  MoveL 5887 to (-63.75, 25.43, -226.45) mm, rotated rx -172.19 ry 6.28 rz 7.52 deg; joints [-6.092, -28.994, 83.557, 94.01, 104.935, 56.545, -36.259]
  MoveL 5888 to (-64.25, 25.28, -226.45) mm, rotated rx -172.19 ry 6.28 rz 7.52 deg; joints [-6.076, -29.01, 83.573, 94.023, 104.926, 56.543, -36.259]
  MoveL 5889 to (-65.23, 24.96, -226.41) mm, rotated rx -172.19 ry 6.28 rz 7.52 deg; joints [-6.045, -29.04, 83.608, 94.048, 104.908, 56.538, -36.259]
  MoveL 5890 to (-67.74, 24.21, -226.41) mm, rotated rx -172.19 ry 6.28 rz 7.52 deg; joints [-5.965, -29.118, 83.687, 94.111, 104.862, 56.533, -36.259]
  MoveL 5891 to (-68.71, 23.85, -226.39) mm, rotated rx -172.19 ry 6.28 rz 7.52 deg; joints [-5.934, -29.151, 83.725, 94.135, 104.844, 56.527, -36.259]
  MoveL 5892 to (-70.09, 23.42, -226.46) mm, rotated rx -172.19 ry 6.28 rz 7.52 deg; joints [-5.891, -29.197, 83.77, 94.17, 104.819, 56.527, -36.259]
  MoveL 5893 to (-71.24, 23.21, -226.71) mm, rotated rx -172.19 ry 6.28 rz 7.52 deg; joints [-5.856, -29.233, 83.787, 94.203, 104.798, 56.544, -36.259]
  MoveL 5894 to (-72.17, 23.22, -227.15) mm, rotated rx -172.19 ry 6.28 rz 7.52 deg; joints [-5.831, -29.259, 83.777, 94.232, 104.781, 56.579, -36.259]
  MoveL 5895 to (-72.55, 23.31, -227.44) mm, rotated rx -172.19 ry 6.28 rz 7.52 deg; joints [-5.822, -29.268, 83.763, 94.245, 104.774, 56.604, -36.259]
  MoveL 5896 to (-72.88, 23.45, -227.78) mm, rotated rx -172.19 ry 6.28 rz 7.52 deg; joints [-5.816, -29.274, 83.741, 94.258, 104.768, 56.632, -36.259]
  MoveL 5897 to (-73.35, 23.9, -228.59) mm, rotated rx -172.19 ry 6.28 rz 7.52 deg; joints [-5.809, -29.28, 83.677, 94.282, 104.759, 56.703, -36.259]
  MoveL 5898 to (-73.61, 24.57, -229.59) mm, rotated rx -172.19 ry 6.28 rz 7.52 deg; joints [-5.812, -29.275, 83.587, 94.302, 104.754, 56.792, -36.259]
  MoveL 5899 to (-73.44, 26.58, -232.15) mm, rotated rx -172.19 ry 6.28 rz 7.52 deg; joints [-5.844, -29.234, 83.324, 94.334, 104.756, 57.022, -36.259]
  MoveL 5900 to (-72.5, 28.79, -234.71) mm, rotated rx -172.19 ry 6.28 rz 7.52 deg; joints [-5.901, -29.171, 83.039, 94.347, 104.773, 57.254, -36.259]
  MoveL 5901 to (-70.94, 30.53, -236.54) mm, rotated rx -172.19 ry 6.28 rz 7.52 deg; joints [-5.97, -29.104, 82.818, 94.333, 104.802, 57.415, -36.259]
  MoveL 5902 to (-69.92, 31.22, -237.18) mm, rotated rx -172.19 ry 6.28 rz 7.52 deg; joints [-6.009, -29.069, 82.733, 94.316, 104.821, 57.469, -36.259]
  MoveL 5903 to (-68.75, 31.79, -237.64) mm, rotated rx -172.19 ry 6.28 rz 7.52 deg; joints [-6.051, -29.034, 82.664, 94.291, 104.843, 57.506, -36.259]
  MoveL 5904 to (-65.94, 32.57, -238.01) mm, rotated rx -172.19 ry 6.28 rz 7.52 deg; joints [-6.144, -28.962, 82.575, 94.221, 104.897, 57.527, -36.259]
  MoveL 5905 to (-62.84, 33.11, -238.01) mm, rotated rx -172.19 ry 6.28 rz 7.52 deg; joints [-6.243, -28.889, 82.52, 94.139, 104.957, 57.514, -36.259]
  MoveL 5906 to (-61.85, 33.31, -238.02) mm, rotated rx -172.19 ry 6.28 rz 7.52 deg; joints [-6.274, -28.865, 82.499, 94.113, 104.976, 57.511, -36.259]
  MoveL 5907 to (-60.81, 33.49, -238.02) mm, rotated rx -172.19 ry 6.28 rz 7.52 deg; joints [-6.307, -28.84, 82.48, 94.085, 104.996, 57.507, -36.259]
  MoveL 5908 to (-60.32, 33.58, -238.02) mm, rotated rx -172.19 ry 6.28 rz 7.52 deg; joints [-6.323, -28.829, 82.471, 94.072, 105.005, 57.505, -36.259]
  MoveL 5909 to (-59.67, 33.7, -238.05) mm, rotated rx -172.19 ry 6.28 rz 7.52 deg; joints [-6.344, -28.814, 82.457, 94.055, 105.018, 57.505, -36.259]
  MoveL 5910 to (-59.09, 33.84, -238.11) mm, rotated rx -172.19 ry 6.28 rz 7.52 deg; joints [-6.363, -28.8, 82.443, 94.04, 105.029, 57.507, -36.259]
  MoveL 5911 to (-58.6, 33.97, -238.18) mm, rotated rx -172.19 ry 6.28 rz 7.52 deg; joints [-6.379, -28.788, 82.427, 94.028, 105.038, 57.511, -36.259]
  MoveL 5912 to (-58.15, 34.08, -238.24) mm, rotated rx -172.19 ry 6.28 rz 7.52 deg; joints [-6.394, -28.777, 82.414, 94.017, 105.047, 57.513, -36.259]
  MoveL 5913 to (-57.7, 34.18, -238.27) mm, rotated rx -172.19 ry 6.28 rz 7.52 deg; joints [-6.409, -28.766, 82.403, 94.005, 105.055, 57.514, -36.259]
  MoveL 5914 to (-56.15, 34.45, -238.27) mm, rotated rx -172.19 ry 6.28 rz 7.52 deg; joints [-6.458, -28.729, 82.375, 93.964, 105.085, 57.508, -36.259]
  MoveL 5915 to (-55.66, 34.56, -238.28) mm, rotated rx -172.19 ry 6.28 rz 7.52 deg; joints [-6.473, -28.716, 82.363, 93.951, 105.094, 57.507, -36.259]
  MoveL 5916 to (-55.23, 34.67, -238.31) mm, rotated rx -172.19 ry 6.28 rz 7.52 deg; joints [-6.487, -28.705, 82.35, 93.941, 105.102, 57.509, -36.259]
  MoveL 5917 to (-54.87, 34.8, -238.36) mm, rotated rx -172.19 ry 6.28 rz 7.52 deg; joints [-6.499, -28.693, 82.335, 93.932, 105.109, 57.514, -36.259]
  MoveL 5918 to (-54.61, 34.96, -238.42) mm, rotated rx -172.19 ry 6.28 rz 7.52 deg; joints [-6.508, -28.682, 82.316, 93.927, 105.114, 57.522, -36.259]
  MoveL 5919 to (-54.41, 35.14, -238.49) mm, rotated rx -172.19 ry 6.28 rz 7.52 deg; joints [-6.515, -28.671, 82.295, 93.924, 105.118, 57.532, -36.259]
  MoveL 5920 to (-55.91, 34.64, -239.3) mm, rotated rx -172.19 ry 6.28 rz 7.52 deg; joints [-6.476, -28.747, 82.338, 93.964, 105.092, 57.565, -36.259]
  MoveL 5921 to (-54.61, 35.83, -239.7) mm, rotated rx -172.19 ry 6.28 rz 7.52 deg; joints [-6.521, -28.669, 82.197, 93.945, 105.115, 57.632, -36.259]
  MoveL 5922 to (-53.25, 37.12, -239.96) mm, rotated rx -172.19 ry 6.28 rz 7.52 deg; joints [-6.566, -28.581, 82.047, 93.926, 105.137, 57.697, -36.259]
  MoveL 5923 to (-51.81, 38.51, -240.15) mm, rotated rx -172.19 ry 6.28 rz 7.52 deg; joints [-6.612, -28.481, 81.886, 93.906, 105.16, 57.763, -36.259]
  MoveL 5924 to (-50.29, 40.01, -240.34) mm, rotated rx -172.19 ry 6.28 rz 7.52 deg; joints [-6.661, -28.375, 81.712, 93.886, 105.185, 57.835, -36.259]
  MoveL 5925 to (-48.76, 41.5, -240.44) mm, rotated rx -172.19 ry 6.28 rz 7.52 deg; joints [-6.709, -28.265, 81.541, 93.865, 105.209, 57.901, -36.259]
  MoveL 5926 to (-47.23, 42.98, -240.53) mm, rotated rx -172.19 ry 6.28 rz 7.52 deg; joints [-6.757, -28.156, 81.369, 93.844, 105.234, 57.967, -36.259]
  MoveL 5927 to (-45.7, 44.48, -240.73) mm, rotated rx -172.19 ry 6.28 rz 7.52 deg; joints [-6.806, -28.049, 81.194, 93.824, 105.258, 58.04, -36.259]
  MoveL 5928 to (-44.17, 45.96, -240.83) mm, rotated rx -172.19 ry 6.28 rz 7.52 deg; joints [-6.854, -27.939, 81.022, 93.803, 105.283, 58.107, -36.259]
  MoveL 5929 to (-42.63, 47.44, -240.93) mm, rotated rx -172.19 ry 6.28 rz 7.52 deg; joints [-6.902, -27.83, 80.849, 93.782, 105.307, 58.174, -36.259]
  MoveL 5930 to (-41.09, 48.92, -241.13) mm, rotated rx -172.19 ry 6.28 rz 7.52 deg; joints [-6.951, -27.723, 80.674, 93.763, 105.332, 58.247, -36.259]
  MoveL 5931 to (-38.01, 51.88, -241.33) mm, rotated rx -172.19 ry 6.28 rz 7.52 deg; joints [-7.046, -27.503, 80.326, 93.722, 105.382, 58.383, -36.259]
  MoveL 5932 to (-36.72, 53.11, -241.54) mm, rotated rx -172.19 ry 6.28 rz 7.52 deg; joints [-7.088, -27.414, 80.178, 93.706, 105.403, 58.446, -36.259]
  MoveL 5933 to (-35.33, 54.5, -241.61) mm, rotated rx -172.19 ry 6.28 rz 7.52 deg; joints [-7.131, -27.31, 80.014, 93.689, 105.425, 58.51, -36.259]
  MoveL 5934 to (-33.91, 55.99, -241.62) mm, rotated rx -172.19 ry 6.28 rz 7.52 deg; joints [-7.173, -27.197, 79.838, 93.673, 105.447, 58.577, -36.259]
  MoveL 5935 to (-31.97, 57.83, -241.73) mm, rotated rx -172.19 ry 6.28 rz 7.52 deg; joints [-7.233, -27.058, 79.619, 93.648, 105.478, 58.662, -36.259]
  MoveL 5936 to (-30.02, 59.52, -241.83) mm, rotated rx -172.19 ry 6.28 rz 7.52 deg; joints [-7.293, -26.928, 79.417, 93.621, 105.509, 58.739, -36.259]
  MoveL 5937 to (-28.4, 61.01, -241.92) mm, rotated rx -172.19 ry 6.28 rz 7.52 deg; joints [-7.343, -26.814, 79.237, 93.6, 105.536, 58.809, -36.259]
  MoveL 5938 to (-26.9, 62.41, -242.1) mm, rotated rx -172.19 ry 6.28 rz 7.52 deg; joints [-7.39, -26.71, 79.067, 93.582, 105.56, 58.879, -36.259]
  MoveL 5939 to (-25.5, 63.7, -242.38) mm, rotated rx -172.19 ry 6.28 rz 7.52 deg; joints [-7.435, -26.617, 78.908, 93.565, 105.583, 58.95, -36.259]
  MoveL 5940 to (-24.11, 64.98, -242.66) mm, rotated rx -172.19 ry 6.28 rz 7.52 deg; joints [-7.479, -26.525, 78.749, 93.549, 105.607, 59.021, -36.259]
  MoveL 5941 to (-22.7, 66.23, -242.96) mm, rotated rx -172.19 ry 6.28 rz 7.52 deg; joints [-7.525, -26.436, 78.594, 93.532, 105.63, 59.09, -36.259]
  MoveL 5942 to (-21.23, 67.57, -243.11) mm, rotated rx -172.19 ry 6.28 rz 7.52 deg; joints [-7.57, -26.334, 78.429, 93.514, 105.654, 59.158, -36.259]
  MoveL 5943 to (-20.58, 67.57, -243.73) mm, rotated rx -172.19 ry 6.28 rz 7.52 deg; joints [-7.597, -26.345, 78.42, 93.499, 105.67, 59.18, -36.259]
  MoveL 5944 to (-20.69, 67.27, -244.04) mm, rotated rx -172.19 ry 6.28 rz 7.52 deg; joints [-7.598, -26.375, 78.451, 93.498, 105.67, 59.179, -36.259]
  MoveL 5945 to (-20.66, 67.23, -244.24) mm, rotated rx -172.19 ry 6.28 rz 7.52 deg; joints [-7.601, -26.383, 78.453, 93.498, 105.671, 59.186, -36.259]
  MoveL 5946 to (-20.52, 67.44, -244.33) mm, rotated rx -172.19 ry 6.28 rz 7.52 deg; joints [-7.606, -26.371, 78.426, 93.498, 105.674, 59.201, -36.259]
  MoveL 5947 to (-20.34, 67.85, -244.35) mm, rotated rx -172.19 ry 6.28 rz 7.52 deg; joints [-7.611, -26.343, 78.376, 93.5, 105.675, 59.223, -36.259]
  MoveL 5948 to (-20.18, 68.31, -244.36) mm, rotated rx -172.19 ry 6.28 rz 7.52 deg; joints [-7.615, -26.311, 78.321, 93.503, 105.676, 59.248, -36.259]
  MoveL 5949 to (-19.97, 69.26, -244.39) mm, rotated rx -172.19 ry 6.28 rz 7.52 deg; joints [-7.621, -26.248, 78.205, 93.514, 105.677, 59.303, -36.259]
  MoveL 5950 to (-19.63, 70.8, -244.39) mm, rotated rx -172.19 ry 6.28 rz 7.52 deg; joints [-7.629, -26.144, 78.019, 93.53, 105.677, 59.388, -36.259]
  MoveL 5951 to (-19.38, 71.74, -244.4) mm, rotated rx -172.19 ry 6.28 rz 7.52 deg; joints [-7.635, -26.081, 77.904, 93.54, 105.677, 59.441, -36.259]
  MoveL 5952 to (-19.16, 72.77, -244.4) mm, rotated rx -172.19 ry 6.28 rz 7.52 deg; joints [-7.64, -26.011, 77.78, 93.551, 105.677, 59.499, -36.259]
  MoveL 5953 to (-19.04, 73.27, -244.42) mm, rotated rx -172.19 ry 6.28 rz 7.52 deg; joints [-7.643, -25.978, 77.719, 93.557, 105.677, 59.528, -36.259]
  MoveL 5954 to (-18.93, 73.73, -244.45) mm, rotated rx -172.19 ry 6.28 rz 7.52 deg; joints [-7.646, -25.948, 77.663, 93.561, 105.678, 59.554, -36.259]
  MoveL 5955 to (-18.81, 74.15, -244.49) mm, rotated rx -172.19 ry 6.28 rz 7.52 deg; joints [-7.65, -25.92, 77.611, 93.566, 105.678, 59.58, -36.259]
  MoveL 5956 to (-18.7, 74.54, -244.56) mm, rotated rx -172.19 ry 6.28 rz 7.52 deg; joints [-7.653, -25.895, 77.562, 93.569, 105.679, 59.605, -36.259]
  MoveL 5957 to (-18.58, 74.94, -244.61) mm, rotated rx -172.19 ry 6.28 rz 7.52 deg; joints [-7.657, -25.869, 77.512, 93.573, 105.68, 59.63, -36.259]
  MoveL 5958 to (-18.46, 75.39, -244.64) mm, rotated rx -172.19 ry 6.28 rz 7.52 deg; joints [-7.66, -25.84, 77.457, 93.578, 105.68, 59.656, -36.259]
  MoveL 5959 to (-18.35, 75.85, -244.67) mm, rotated rx -172.19 ry 6.28 rz 7.52 deg; joints [-7.663, -25.809, 77.4, 93.583, 105.68, 59.683, -36.259]
  MoveL 5960 to (-18.22, 76.27, -244.71) mm, rotated rx -172.19 ry 6.28 rz 7.52 deg; joints [-7.667, -25.781, 77.349, 93.587, 105.681, 59.709, -36.259]
  MoveL 5961 to (-18.1, 76.65, -244.77) mm, rotated rx -172.19 ry 6.28 rz 7.52 deg; joints [-7.671, -25.757, 77.301, 93.59, 105.682, 59.733, -36.259]
  MoveL 5962 to (-17.98, 77.04, -244.82) mm, rotated rx -172.19 ry 6.28 rz 7.52 deg; joints [-7.674, -25.731, 77.252, 93.594, 105.683, 59.757, -36.259]
  MoveL 5963 to (-17.86, 77.47, -244.85) mm, rotated rx -172.19 ry 6.28 rz 7.52 deg; joints [-7.678, -25.703, 77.2, 93.598, 105.683, 59.782, -36.259]
  MoveL 5964 to (-17.75, 77.98, -244.85) mm, rotated rx -172.19 ry 6.28 rz 7.52 deg; joints [-7.68, -25.668, 77.137, 93.604, 105.683, 59.811, -36.259]
  MoveL 5965 to (-16.88, 80.76, -245.21) mm, rotated rx -172.19 ry 6.28 rz 7.52 deg; joints [-7.707, -25.485, 76.79, 93.63, 105.689, 59.983, -36.259]
  MoveL 5966 to (-16.3, 81.92, -245.65) mm, rotated rx -172.19 ry 6.28 rz 7.52 deg; joints [-7.727, -25.416, 76.64, 93.637, 105.697, 60.067, -36.259]
  MoveL 5967 to (-15.62, 82.91, -246.28) mm, rotated rx -172.19 ry 6.28 rz 7.52 deg; joints [-7.753, -25.36, 76.507, 93.639, 105.708, 60.148, -36.259]
  MoveL 5968 to (-13.99, 84.42, -248.06) mm, rotated rx -172.19 ry 6.28 rz 7.52 deg; joints [-7.82, -25.293, 76.29, 93.629, 105.741, 60.306, -36.259]
  MoveL 5969 to (-11.99, 85.29, -250.55) mm, rotated rx -172.19 ry 6.28 rz 7.52 deg; joints [-7.907, -25.283, 76.139, 93.603, 105.786, 60.456, -36.259]
  MoveL 5970 to (-10.19, 85.39, -253.05) mm, rotated rx -172.19 ry 6.28 rz 7.52 deg; joints [-7.988, -25.326, 76.082, 93.569, 105.832, 60.563, -36.259]
  MoveL 5971 to (-9.6, 85.11, -254.02) mm, rotated rx -172.19 ry 6.28 rz 7.52 deg; joints [-8.017, -25.365, 76.099, 93.553, 105.849, 60.587, -36.259]
  MoveL 5972 to (-9.2, 84.61, -254.83) mm, rotated rx -172.19 ry 6.28 rz 7.52 deg; joints [-8.039, -25.417, 76.147, 93.538, 105.862, 60.592, -36.259]
  MoveL 5973 to (-9.08, 84.28, -255.16) mm, rotated rx -172.19 ry 6.28 rz 7.52 deg; joints [-8.047, -25.447, 76.183, 93.53, 105.867, 60.587, -36.259]
  MoveL 5974 to (-9.01, 83.89, -255.45) mm, rotated rx -172.19 ry 6.28 rz 7.52 deg; joints [-8.052, -25.48, 76.226, 93.523, 105.872, 60.577, -36.259]
  MoveL 5975 to (-9.02, 82.94, -255.89) mm, rotated rx -172.19 ry 6.28 rz 7.52 deg; joints [-8.059, -25.556, 76.335, 93.509, 105.877, 60.542, -36.259]
  MoveL 5976 to (-9.23, 81.77, -256.16) mm, rotated rx -172.19 ry 6.28 rz 7.52 deg; joints [-8.057, -25.644, 76.475, 93.495, 105.88, 60.488, -36.259]
  MoveL 5977 to (-9.65, 80.38, -256.25) mm, rotated rx -172.19 ry 6.28 rz 7.52 deg; joints [-8.048, -25.744, 76.645, 93.482, 105.878, 60.414, -36.259]
  MoveL 5978 to (-10.5, 77.9, -256.25) mm, rotated rx -172.19 ry 6.28 rz 7.52 deg; joints [-8.026, -25.918, 76.951, 93.462, 105.872, 60.277, -36.259]
  MoveL 5979 to (-10.65, 77.49, -256.22) mm, rotated rx -172.19 ry 6.28 rz 7.52 deg; joints [-8.021, -25.946, 77.002, 93.458, 105.871, 60.253, -36.259]
  MoveL 5980 to (-10.81, 77.12, -256.17) mm, rotated rx -172.19 ry 6.28 rz 7.52 deg; joints [-8.017, -25.971, 77.048, 93.456, 105.869, 60.231, -36.259]
  MoveL 5981 to (-10.97, 76.77, -256.1) mm, rotated rx -172.19 ry 6.28 rz 7.52 deg; joints [-8.012, -25.994, 77.093, 93.454, 105.867, 60.208, -36.259]
  MoveL 5982 to (-11.13, 76.37, -256.05) mm, rotated rx -172.19 ry 6.28 rz 7.52 deg; joints [-8.007, -26.021, 77.142, 93.451, 105.866, 60.184, -36.259]
  MoveL 5983 to (-11.31, 75.9, -256.01) mm, rotated rx -172.19 ry 6.28 rz 7.52 deg; joints [-8.002, -26.053, 77.2, 93.447, 105.864, 60.157, -36.259]
  MoveL 5984 to (-11.51, 75.42, -255.96) mm, rotated rx -172.19 ry 6.28 rz 7.52 deg; joints [-7.996, -26.085, 77.261, 93.444, 105.862, 60.128, -36.259]
  MoveL 5985 to (-11.69, 74.91, -255.94) mm, rotated rx -172.19 ry 6.28 rz 7.52 deg; joints [-7.991, -26.121, 77.324, 93.44, 105.861, 60.099, -36.259]
  MoveL 5986 to (-11.9, 74.3, -255.96) mm, rotated rx -172.19 ry 6.28 rz 7.52 deg; joints [-7.986, -26.163, 77.398, 93.435, 105.859, 60.067, -36.259]
  MoveL 5987 to (-12.15, 73.47, -256.02) mm, rotated rx -172.19 ry 6.28 rz 7.52 deg; joints [-7.98, -26.223, 77.498, 93.428, 105.858, 60.024, -36.259]
  MoveL 5988 to (-12.32, 72.97, -256.02) mm, rotated rx -172.19 ry 6.28 rz 7.52 deg; joints [-7.976, -26.258, 77.558, 93.424, 105.857, 59.997, -36.259]
  MoveL 5989 to (-12.49, 72.5, -256.01) mm, rotated rx -172.19 ry 6.28 rz 7.52 deg; joints [-7.971, -26.29, 77.616, 93.42, 105.856, 59.971, -36.259]
  MoveL 5990 to (-12.65, 72.06, -255.99) mm, rotated rx -172.19 ry 6.28 rz 7.52 deg; joints [-7.967, -26.32, 77.67, 93.417, 105.854, 59.947, -36.259]
  MoveL 5991 to (-12.81, 71.68, -255.94) mm, rotated rx -172.19 ry 6.28 rz 7.52 deg; joints [-7.962, -26.346, 77.717, 93.415, 105.853, 59.924, -36.259]
  MoveL 5992 to (-12.98, 71.32, -255.88) mm, rotated rx -172.19 ry 6.28 rz 7.52 deg; joints [-7.957, -26.37, 77.762, 93.413, 105.851, 59.902, -36.259]
  MoveL 5993 to (-13.2, 70.96, -255.83) mm, rotated rx -172.19 ry 6.28 rz 7.52 deg; joints [-7.95, -26.395, 77.807, 93.412, 105.848, 59.881, -36.259]
  MoveL 5994 to (-13.45, 70.63, -255.78) mm, rotated rx -172.19 ry 6.28 rz 7.52 deg; joints [-7.942, -26.417, 77.848, 93.413, 105.844, 59.862, -36.259]
  MoveL 5995 to (-13.63, 70.5, -255.61) mm, rotated rx -172.19 ry 6.28 rz 7.52 deg; joints [-7.935, -26.424, 77.867, 93.415, 105.84, 59.848, -36.259]
  MoveL 5996 to (-13.63, 70.61, -255.3) mm, rotated rx -172.19 ry 6.28 rz 7.52 deg; joints [-7.931, -26.407, 77.859, 93.415, 105.838, 59.839, -36.259]
  MoveL 5997 to (-13.43, 71, -254.81) mm, rotated rx -172.19 ry 6.28 rz 7.52 deg; joints [-7.932, -26.364, 77.82, 93.414, 105.839, 59.835, -36.259]
  MoveL 5998 to (-14.11, 70.43, -253.96) mm, rotated rx -172.19 ry 6.28 rz 7.52 deg; joints [-7.903, -26.385, 77.903, 93.419, 105.824, 59.769, -36.259]
  MoveL 5999 to (-17.51, 67.85, -253.96) mm, rotated rx -172.19 ry 6.28 rz 7.52 deg; joints [-7.801, -26.598, 78.219, 93.468, 105.768, 59.659, -36.259]
  MoveL 6000 to (-19.11, 66.64, -253.89) mm, rotated rx -172.19 ry 6.28 rz 7.52 deg; joints [-7.752, -26.696, 78.367, 93.492, 105.74, 59.605, -36.259]
  MoveL 6001 to (-20.7, 65.45, -253.74) mm, rotated rx -172.19 ry 6.28 rz 7.52 deg; joints [-7.703, -26.79, 78.514, 93.515, 105.713, 59.548, -36.259]
  MoveL 6002 to (-22.54, 64.08, -253.55) mm, rotated rx -172.19 ry 6.28 rz 7.52 deg; joints [-7.645, -26.897, 78.683, 93.543, 105.681, 59.482, -36.259]
  MoveL 6003 to (-24.28, 62.78, -253.33) mm, rotated rx -172.19 ry 6.28 rz 7.52 deg; joints [-7.591, -26.998, 78.843, 93.568, 105.651, 59.418, -36.259]
  MoveL 6004 to (-26.02, 61.46, -253.23) mm, rotated rx -172.19 ry 6.28 rz 7.52 deg; joints [-7.537, -27.103, 79.002, 93.595, 105.622, 59.359, -36.259]
  MoveL 6005 to (-27.72, 60.17, -253.23) mm, rotated rx -172.19 ry 6.28 rz 7.52 deg; joints [-7.486, -27.208, 79.157, 93.621, 105.593, 59.306, -36.259]
  MoveL 6006 to (-29.3, 58.97, -253.17) mm, rotated rx -172.19 ry 6.28 rz 7.52 deg; joints [-7.437, -27.305, 79.302, 93.645, 105.566, 59.254, -36.259]
  MoveL 6007 to (-30.79, 57.83, -253.05) mm, rotated rx -172.19 ry 6.28 rz 7.52 deg; joints [-7.391, -27.394, 79.439, 93.668, 105.541, 59.202, -36.259]
  MoveL 6008 to (-32.42, 56.59, -252.98) mm, rotated rx -172.19 ry 6.28 rz 7.52 deg; joints [-7.341, -27.492, 79.587, 93.693, 105.514, 59.149, -36.259]
  MoveL 6009 to (-34.11, 55.3, -252.8) mm, rotated rx -172.19 ry 6.28 rz 7.52 deg; joints [-7.288, -27.592, 79.743, 93.719, 105.485, 59.089, -36.259]
  MoveL 6010 to (-37.51, 52.71, -252.62) mm, rotated rx -172.19 ry 6.28 rz 7.52 deg; joints [-7.182, -27.796, 80.05, 93.772, 105.427, 58.977, -36.259]
  MoveL 6011 to (-39.2, 51.41, -252.44) mm, rotated rx -172.19 ry 6.28 rz 7.52 deg; joints [-7.129, -27.895, 80.205, 93.799, 105.398, 58.917, -36.259]
  MoveL 6012 to (-40.89, 50.1, -252.26) mm, rotated rx -172.19 ry 6.28 rz 7.52 deg; joints [-7.075, -27.995, 80.361, 93.825, 105.369, 58.857, -36.259]
  MoveL 6013 to (-42.58, 48.81, -252.26) mm, rotated rx -172.19 ry 6.28 rz 7.52 deg; joints [-7.023, -28.098, 80.511, 93.853, 105.341, 58.807, -36.259]
  MoveL 6014 to (-44.27, 47.5, -252.08) mm, rotated rx -172.19 ry 6.28 rz 7.52 deg; joints [-6.97, -28.198, 80.666, 93.879, 105.312, 58.747, -36.259]
  MoveL 6015 to (-45.95, 46.19, -251.91) mm, rotated rx -172.19 ry 6.28 rz 7.52 deg; joints [-6.917, -28.297, 80.82, 93.906, 105.283, 58.688, -36.259]
  MoveL 6016 to (-47.65, 44.9, -251.91) mm, rotated rx -172.19 ry 6.28 rz 7.52 deg; joints [-6.864, -28.4, 80.969, 93.935, 105.255, 58.639, -36.259]
  MoveL 6017 to (-49.16, 43.66, -251.71) mm, rotated rx -172.19 ry 6.28 rz 7.52 deg; joints [-6.816, -28.492, 81.114, 93.958, 105.229, 58.581, -36.259]
  MoveL 6018 to (-50.44, 42.52, -251.39) mm, rotated rx -172.19 ry 6.28 rz 7.52 deg; joints [-6.773, -28.569, 81.25, 93.976, 105.207, 58.519, -36.259]
  MoveL 6019 to (-51.53, 41.45, -250.93) mm, rotated rx -172.19 ry 6.28 rz 7.52 deg; joints [-6.735, -28.636, 81.38, 93.988, 105.188, 58.452, -36.259]
  MoveL 6020 to (-50.68, 41.87, -250.16) mm, rotated rx -172.19 ry 6.28 rz 7.52 deg; joints [-6.753, -28.575, 81.344, 93.967, 105.201, 58.426, -36.259]
  MoveL 6021 to (-51.03, 41.66, -250.15) mm, rotated rx -172.19 ry 6.28 rz 7.52 deg; joints [-6.742, -28.592, 81.368, 93.974, 105.195, 58.419, -36.259]
  MoveC 6022 to (-54.55, 41.16, -250.15) mm, rotated rx -172.19 ry 6.28 rz 7.52 deg; joints [-6.631, -28.669, 81.421, 94.068, 105.126, 58.438, -36.259] to (-58.1, 40.96, -250.15) mm, rotated rx -172.19 ry 6.28 rz 7.52 deg; joints [-6.519, -28.728, 81.439, 94.167, 105.055, 58.475, -36.259]
  MoveL 6023 to (-58.1, 40.96, -250.15) mm, rotated rx -172.19 ry 6.28 rz 7.52 deg; joints [-6.519, -28.728, 81.439, 94.167, 105.055, 58.475, -36.259]
  MoveL 6024 to (-58.57, 40.92, -250.13) mm, rotated rx -172.19 ry 6.28 rz 7.52 deg; joints [-6.504, -28.735, 81.443, 94.18, 105.046, 58.478, -36.259]
  MoveL 6025 to (-58.99, 40.87, -250.08) mm, rotated rx -172.19 ry 6.28 rz 7.52 deg; joints [-6.49, -28.742, 81.45, 94.191, 105.038, 58.478, -36.259]
  MoveL 6026 to (-59.39, 40.81, -250.02) mm, rotated rx -172.19 ry 6.28 rz 7.52 deg; joints [-6.476, -28.749, 81.457, 94.201, 105.03, 58.478, -36.259]
  MoveL 6027 to (-59.83, 40.76, -249.97) mm, rotated rx -172.19 ry 6.28 rz 7.52 deg; joints [-6.462, -28.757, 81.462, 94.213, 105.021, 58.479, -36.259]
  MoveL 6028 to (-60.3, 40.71, -249.95) mm, rotated rx -172.19 ry 6.28 rz 7.52 deg; joints [-6.447, -28.765, 81.467, 94.225, 105.011, 58.481, -36.259]
  MoveL 6029 to (-60.82, 40.67, -249.93) mm, rotated rx -172.19 ry 6.28 rz 7.52 deg; joints [-6.43, -28.773, 81.471, 94.24, 105.001, 58.485, -36.259]
  MoveL 6030 to (-61.86, 40.61, -249.93) mm, rotated rx -172.19 ry 6.28 rz 7.52 deg; joints [-6.397, -28.79, 81.476, 94.269, 104.98, 58.496, -36.259]
  MoveL 6031 to (-63.32, 40.58, -250.02) mm, rotated rx -172.19 ry 6.28 rz 7.52 deg; joints [-6.352, -28.813, 81.475, 94.31, 104.951, 58.519, -36.259]
  MoveL 6032 to (-64.51, 40.68, -250.3) mm, rotated rx -172.19 ry 6.28 rz 7.52 deg; joints [-6.317, -28.831, 81.456, 94.348, 104.927, 58.555, -36.259]
  MoveL 6033 to (-65.45, 40.91, -250.75) mm, rotated rx -172.19 ry 6.28 rz 7.52 deg; joints [-6.292, -28.842, 81.42, 94.38, 104.908, 58.603, -36.259]
  MoveL 6034 to (-66.13, 41.27, -251.39) mm, rotated rx -172.19 ry 6.28 rz 7.52 deg; joints [-6.277, -28.848, 81.367, 94.407, 104.895, 58.663, -36.259]
  MoveL 6035 to (-66.56, 41.76, -252.22) mm, rotated rx -172.19 ry 6.28 rz 7.52 deg; joints [-6.272, -28.849, 81.296, 94.43, 104.886, 58.737, -36.259]
  MoveL 6036 to (-66.72, 42.39, -253.22) mm, rotated rx -172.19 ry 6.28 rz 7.52 deg; joints [-6.277, -28.843, 81.207, 94.448, 104.883, 58.823, -36.259]
  MoveL 6037 to (-66.28, 44.02, -255.78) mm, rotated rx -172.19 ry 6.28 rz 7.52 deg; joints [-6.318, -28.814, 80.977, 94.47, 104.892, 59.033, -36.259]
  MoveL 6038 to (-65.04, 45.65, -258.34) mm, rotated rx -172.19 ry 6.28 rz 7.52 deg; joints [-6.383, -28.775, 80.747, 94.47, 104.917, 59.232, -36.259]
  MoveL 6039 to (-64.21, 46.28, -259.35) mm, rotated rx -172.19 ry 6.28 rz 7.52 deg; joints [-6.42, -28.755, 80.659, 94.46, 104.934, 59.305, -36.259]
  MoveL 6040 to (-63.25, 46.78, -260.17) mm, rotated rx -172.19 ry 6.28 rz 7.52 deg; joints [-6.459, -28.737, 80.589, 94.443, 104.954, 59.36, -36.259]
  MoveL 6041 to (-62.15, 47.15, -260.81) mm, rotated rx -172.19 ry 6.28 rz 7.52 deg; joints [-6.5, -28.719, 80.537, 94.42, 104.977, 59.398, -36.259]
  MoveL 6042 to (-60.9, 47.39, -261.27) mm, rotated rx -172.19 ry 6.28 rz 7.52 deg; joints [-6.544, -28.702, 80.503, 94.391, 105.003, 59.417, -36.259]
  MoveL 6043 to (-58.01, 47.49, -261.63) mm, rotated rx -172.19 ry 6.28 rz 7.52 deg; joints [-6.639, -28.671, 80.491, 94.312, 105.063, 59.402, -36.259]
  MoveL 6044 to (-56.96, 47.44, -261.63) mm, rotated rx -172.19 ry 6.28 rz 7.52 deg; joints [-6.672, -28.661, 80.499, 94.282, 105.085, 59.385, -36.259]
  MoveL 6045 to (-56.44, 47.42, -261.64) mm, rotated rx -172.19 ry 6.28 rz 7.52 deg; joints [-6.689, -28.656, 80.502, 94.267, 105.096, 59.377, -36.259]
  MoveL 6046 to (-55.96, 47.41, -261.66) mm, rotated rx -172.19 ry 6.28 rz 7.52 deg; joints [-6.704, -28.651, 80.503, 94.253, 105.105, 59.371, -36.259]
  MoveL 6047 to (-55.54, 47.41, -261.71) mm, rotated rx -172.19 ry 6.28 rz 7.52 deg; joints [-6.718, -28.646, 80.502, 94.241, 105.114, 59.368, -36.259]
  MoveL 6048 to (-55.14, 47.42, -261.77) mm, rotated rx -172.19 ry 6.28 rz 7.52 deg; joints [-6.731, -28.642, 80.501, 94.23, 105.123, 59.366, -36.259]
  MoveL 6049 to (-54.72, 47.43, -261.82) mm, rotated rx -172.19 ry 6.28 rz 7.52 deg; joints [-6.745, -28.638, 80.5, 94.219, 105.131, 59.363, -36.259]
  MoveL 6050 to (-54.25, 47.42, -261.84) mm, rotated rx -172.19 ry 6.28 rz 7.52 deg; joints [-6.76, -28.633, 80.502, 94.206, 105.141, 59.358, -36.259]
  MoveL 6051 to (-53.75, 47.4, -261.84) mm, rotated rx -172.19 ry 6.28 rz 7.52 deg; joints [-6.776, -28.629, 80.505, 94.191, 105.151, 59.35, -36.259]
  MoveL 6052 to (-53.2, 47.37, -261.84) mm, rotated rx -172.19 ry 6.28 rz 7.52 deg; joints [-6.793, -28.623, 80.509, 94.175, 105.163, 59.341, -36.259]
  MoveL 6053 to (-52.67, 47.35, -261.84) mm, rotated rx -172.19 ry 6.28 rz 7.52 deg; joints [-6.81, -28.618, 80.512, 94.16, 105.174, 59.333, -36.259]
  MoveL 6054 to (-52.18, 47.33, -261.87) mm, rotated rx -172.19 ry 6.28 rz 7.52 deg; joints [-6.826, -28.613, 80.514, 94.146, 105.184, 59.327, -36.259]
  MoveL 6055 to (-51.7, 47.33, -261.91) mm, rotated rx -172.19 ry 6.28 rz 7.52 deg; joints [-6.841, -28.609, 80.514, 94.132, 105.194, 59.323, -36.259]
  MoveL 6056 to (-51.2, 47.34, -261.99) mm, rotated rx -172.19 ry 6.28 rz 7.52 deg; joints [-6.858, -28.604, 80.512, 94.119, 105.204, 59.321, -36.259]
  MoveL 6057 to (-50.59, 47.35, -262.05) mm, rotated rx -172.19 ry 6.28 rz 7.52 deg; joints [-6.878, -28.597, 80.511, 94.102, 105.217, 59.316, -36.259]
  MoveL 6058 to (-50.02, 47.34, -262.07) mm, rotated rx -172.19 ry 6.28 rz 7.52 deg; joints [-6.896, -28.591, 80.513, 94.086, 105.229, 59.309, -36.259]
  MoveL 6059 to (-49.49, 47.31, -262.07) mm, rotated rx -172.19 ry 6.28 rz 7.52 deg; joints [-6.913, -28.586, 80.516, 94.07, 105.24, 59.301, -36.259]
  MoveL 6060 to (-48.97, 47.29, -262.07) mm, rotated rx -172.19 ry 6.28 rz 7.52 deg; joints [-6.929, -28.581, 80.52, 94.055, 105.25, 59.292, -36.259]
  MoveL 6061 to (-48.31, 47.28, -262.08) mm, rotated rx -172.19 ry 6.28 rz 7.52 deg; joints [-6.95, -28.573, 80.522, 94.036, 105.264, 59.284, -36.259]
  MoveL 6062 to (-47.73, 47.29, -262.09) mm, rotated rx -172.19 ry 6.28 rz 7.52 deg; joints [-6.969, -28.566, 80.521, 94.02, 105.276, 59.277, -36.259]
  MoveL 6063 to (-47.22, 47.32, -262.1) mm, rotated rx -172.19 ry 6.28 rz 7.52 deg; joints [-6.985, -28.557, 80.518, 94.006, 105.286, 59.272, -36.259]
  MoveL 6064 to (-46.89, 47.4, -262.1) mm, rotated rx -172.19 ry 6.28 rz 7.52 deg; joints [-6.995, -28.548, 80.509, 93.998, 105.292, 59.272, -36.259]
  MoveL 6065 to (-46.64, 47.5, -262.1) mm, rotated rx -172.19 ry 6.28 rz 7.52 deg; joints [-7.003, -28.538, 80.497, 93.992, 105.297, 59.275, -36.259]
  MoveL 6066 to (-47.5, 47.13, -262.69) mm, rotated rx -172.19 ry 6.28 rz 7.52 deg; joints [-6.983, -28.591, 80.529, 94.014, 105.283, 59.295, -36.259]
  MoveL 6067 to (-46.52, 48.04, -263.22) mm, rotated rx -172.19 ry 6.28 rz 7.52 deg; joints [-7.018, -28.537, 80.415, 94.003, 105.301, 59.359, -36.259]
  MoveL 6068 to (-45.29, 48.99, -263.61) mm, rotated rx -172.19 ry 6.28 rz 7.52 deg; joints [-7.06, -28.472, 80.298, 93.985, 105.323, 59.415, -36.259]
  MoveL 6069 to (-43.76, 50.03, -263.86) mm, rotated rx -172.19 ry 6.28 rz 7.52 deg; joints [-7.109, -28.394, 80.173, 93.959, 105.35, 59.465, -36.259]
  MoveL 6070 to (-42.02, 51.12, -263.99) mm, rotated rx -172.19 ry 6.28 rz 7.52 deg; joints [-7.164, -28.306, 80.045, 93.928, 105.381, 59.509, -36.259]
  MoveL 6071 to (-40.22, 52.21, -264.08) mm, rotated rx -172.19 ry 6.28 rz 7.52 deg; joints [-7.22, -28.215, 79.915, 93.895, 105.413, 59.552, -36.259]
  MoveL 6072 to (-36.58, 54.43, -264.26) mm, rotated rx -172.19 ry 6.28 rz 7.52 deg; joints [-7.334, -28.031, 79.653, 93.829, 105.478, 59.638, -36.259]
  MoveL 6073 to (-34.76, 55.54, -264.44) mm, rotated rx -172.19 ry 6.28 rz 7.52 deg; joints [-7.391, -27.941, 79.518, 93.797, 105.511, 59.687, -36.259]
  MoveL 6074 to (-31.11, 57.75, -264.62) mm, rotated rx -172.19 ry 6.28 rz 7.52 deg; joints [-7.504, -27.756, 79.254, 93.732, 105.576, 59.774, -36.259]
  MoveL 6075 to (-29.28, 58.86, -264.8) mm, rotated rx -172.19 ry 6.28 rz 7.52 deg; joints [-7.562, -27.666, 79.119, 93.7, 105.609, 59.823, -36.259]
  MoveL 6076 to (-27.45, 59.96, -264.89) mm, rotated rx -172.19 ry 6.28 rz 7.52 deg; joints [-7.618, -27.573, 78.986, 93.668, 105.641, 59.867, -36.259]
  MoveL 6077 to (-25.75, 60.96, -265.11) mm, rotated rx -172.19 ry 6.28 rz 7.52 deg; joints [-7.672, -27.492, 78.862, 93.638, 105.672, 59.913, -36.259]
  MoveL 6078 to (-23.73, 62.17, -265.25) mm, rotated rx -172.19 ry 6.28 rz 7.52 deg; joints [-7.735, -27.391, 78.714, 93.603, 105.708, 59.965, -36.259]
  MoveL 6079 to (-21.53, 63.5, -265.37) mm, rotated rx -172.19 ry 6.28 rz 7.52 deg; joints [-7.803, -27.279, 78.552, 93.565, 105.747, 60.02, -36.259]
  MoveL 6080 to (-19.71, 64.6, -265.37) mm, rotated rx -172.19 ry 6.28 rz 7.52 deg; joints [-7.858, -27.183, 78.418, 93.533, 105.78, 60.061, -36.259]
  MoveL 6081 to (-17.96, 65.64, -265.45) mm, rotated rx -172.19 ry 6.28 rz 7.52 deg; joints [-7.912, -27.094, 78.29, 93.503, 105.811, 60.104, -36.259]
  MoveL 6082 to (-16.38, 66.56, -265.62) mm, rotated rx -172.19 ry 6.28 rz 7.52 deg; joints [-7.961, -27.018, 78.174, 93.476, 105.839, 60.146, -36.259]
  MoveL 6083 to (-14.76, 67.5, -265.83) mm, rotated rx -172.19 ry 6.28 rz 7.52 deg; joints [-8.013, -26.941, 78.057, 93.448, 105.869, 60.191, -36.259]
  MoveL 6084 to (-12.73, 68.7, -265.97) mm, rotated rx -172.19 ry 6.28 rz 7.52 deg; joints [-8.075, -26.839, 77.906, 93.414, 105.905, 60.244, -36.259]
  MoveL 6085 to (-10.52, 70.02, -266.07) mm, rotated rx -172.19 ry 6.28 rz 7.52 deg; joints [-8.143, -26.725, 77.741, 93.377, 105.945, 60.3, -36.259]
  MoveL 6086 to (-6.86, 72.22, -266.07) mm, rotated rx -172.19 ry 6.28 rz 7.52 deg; joints [-8.253, -26.531, 77.468, 93.315, 106.009, 60.385, -36.259]
  MoveL 6087 to (-6.56, 72.13, -266.77) mm, rotated rx -172.19 ry 6.28 rz 7.52 deg; joints [-8.269, -26.553, 77.467, 93.309, 106.018, 60.411, -36.259]
  MoveL 6088 to (-6.74, 71.88, -267.11) mm, rotated rx -172.19 ry 6.28 rz 7.52 deg; joints [-8.268, -26.583, 77.492, 93.311, 106.017, 60.415, -36.259]
  MoveL 6089 to (-6.73, 71.86, -267.33) mm, rotated rx -172.19 ry 6.28 rz 7.52 deg; joints [-8.27, -26.59, 77.49, 93.312, 106.018, 60.425, -36.259]
  MoveL 6090 to (-6.56, 72.06, -267.44) mm, rotated rx -172.19 ry 6.28 rz 7.52 deg; joints [-8.276, -26.578, 77.463, 93.312, 106.021, 60.44, -36.259]
  MoveL 6091 to (-6.32, 72.44, -267.47) mm, rotated rx -172.19 ry 6.28 rz 7.52 deg; joints [-8.284, -26.551, 77.416, 93.312, 106.024, 60.461, -36.259]
  MoveL 6092 to (-6.08, 72.86, -267.5) mm, rotated rx -172.19 ry 6.28 rz 7.52 deg; joints [-8.29, -26.521, 77.364, 93.313, 106.027, 60.484, -36.259]
  MoveL 6093 to (-5.88, 73.24, -267.55) mm, rotated rx -172.19 ry 6.28 rz 7.52 deg; joints [-8.297, -26.495, 77.317, 93.314, 106.03, 60.506, -36.259]
  MoveL 6094 to (-5.68, 73.59, -267.62) mm, rotated rx -172.19 ry 6.28 rz 7.52 deg; joints [-8.303, -26.471, 77.273, 93.315, 106.033, 60.528, -36.259]
  MoveL 6095 to (-5.48, 73.95, -267.67) mm, rotated rx -172.19 ry 6.28 rz 7.52 deg; joints [-8.309, -26.447, 77.228, 93.317, 106.036, 60.549, -36.259]
  MoveL 6096 to (-5.27, 74.34, -267.71) mm, rotated rx -172.19 ry 6.28 rz 7.52 deg; joints [-8.315, -26.419, 77.179, 93.318, 106.038, 60.572, -36.259]
  MoveL 6097 to (-5.04, 74.81, -267.74) mm, rotated rx -172.19 ry 6.28 rz 7.52 deg; joints [-8.321, -26.386, 77.121, 93.32, 106.041, 60.598, -36.259]
  MoveL 6098 to (-4.79, 75.28, -267.8) mm, rotated rx -172.19 ry 6.28 rz 7.52 deg; joints [-8.329, -26.354, 77.062, 93.322, 106.044, 60.626, -36.259]
  MoveL 6099 to (-4.55, 75.74, -267.83) mm, rotated rx -172.19 ry 6.28 rz 7.52 deg; joints [-8.336, -26.321, 77.004, 93.324, 106.047, 60.652, -36.259]
  MoveL 6100 to (-4.33, 76.21, -267.84) mm, rotated rx -172.19 ry 6.28 rz 7.52 deg; joints [-8.342, -26.287, 76.947, 93.326, 106.049, 60.677, -36.259]
  MoveL 6101 to (-4.11, 76.68, -267.84) mm, rotated rx -172.19 ry 6.28 rz 7.52 deg; joints [-8.348, -26.253, 76.888, 93.329, 106.052, 60.703, -36.259]
  MoveL 6102 to (-3.83, 77.31, -267.8) mm, rotated rx -172.19 ry 6.28 rz 7.52 deg; joints [-8.355, -26.206, 76.811, 93.332, 106.054, 60.735, -36.259]
  MoveL 6103 to (-3.56, 77.92, -267.77) mm, rotated rx -172.19 ry 6.28 rz 7.52 deg; joints [-8.361, -26.162, 76.736, 93.336, 106.057, 60.766, -36.259]
  MoveL 6104 to (-3.31, 78.47, -267.77) mm, rotated rx -172.19 ry 6.28 rz 7.52 deg; joints [-8.368, -26.122, 76.669, 93.339, 106.059, 60.795, -36.259]
  MoveL 6105 to (-3.09, 78.88, -267.8) mm, rotated rx -172.19 ry 6.28 rz 7.52 deg; joints [-8.374, -26.093, 76.617, 93.341, 106.062, 60.819, -36.259]
  MoveL 6106 to (-2.89, 79.24, -267.86) mm, rotated rx -172.19 ry 6.28 rz 7.52 deg; joints [-8.381, -26.068, 76.571, 93.342, 106.065, 60.841, -36.259]
  MoveL 6107 to (-2.69, 79.6, -267.92) mm, rotated rx -172.19 ry 6.28 rz 7.52 deg; joints [-8.387, -26.043, 76.526, 93.343, 106.067, 60.863, -36.259]
  MoveL 6108 to (-2.49, 79.99, -267.95) mm, rotated rx -172.19 ry 6.28 rz 7.52 deg; joints [-8.392, -26.016, 76.477, 93.345, 106.07, 60.885, -36.259]
  MoveL 6109 to (-1.82, 81.41, -267.95) mm, rotated rx -172.19 ry 6.28 rz 7.52 deg; joints [-8.41, -25.912, 76.3, 93.353, 106.077, 60.962, -36.259]
  MoveL 6110 to (-0.39, 83.93, -268.33) mm, rotated rx -172.19 ry 6.28 rz 7.52 deg; joints [-8.453, -25.737, 75.98, 93.362, 106.096, 61.115, -36.259]
  MoveL 6111 to (0.39, 84.91, -268.8) mm, rotated rx -172.19 ry 6.28 rz 7.52 deg; joints [-8.48, -25.674, 75.847, 93.361, 106.109, 61.188, -36.259]
  MoveL 6112 to (1.2, 85.71, -269.46) mm, rotated rx -172.19 ry 6.28 rz 7.52 deg; joints [-8.51, -25.629, 75.734, 93.358, 106.124, 61.26, -36.259]
  MoveL 6113 to (2.06, 86.33, -270.31) mm, rotated rx -172.19 ry 6.28 rz 7.52 deg; joints [-8.544, -25.6, 75.639, 93.351, 106.142, 61.329, -36.259]
  MoveL 6114 to (2.96, 86.77, -271.34) mm, rotated rx -172.19 ry 6.28 rz 7.52 deg; joints [-8.582, -25.588, 75.564, 93.341, 106.163, 61.397, -36.259]
  MoveL 6115 to (4.88, 87.11, -273.98) mm, rotated rx -172.19 ry 6.28 rz 7.52 deg; joints [-8.668, -25.615, 75.469, 93.312, 106.211, 61.527, -36.259]
  MoveL 6116 to (6.42, 86.74, -276.62) mm, rotated rx -172.19 ry 6.28 rz 7.52 deg; joints [-8.743, -25.693, 75.461, 93.28, 106.254, 61.619, -36.259]
  MoveL 6117 to (6.86, 86.31, -277.65) mm, rotated rx -172.19 ry 6.28 rz 7.52 deg; joints [-8.768, -25.745, 75.495, 93.267, 106.269, 61.64, -36.259]
  MoveL 6118 to (7.06, 85.7, -278.5) mm, rotated rx -172.19 ry 6.28 rz 7.52 deg; joints [-8.785, -25.807, 75.553, 93.255, 106.28, 61.643, -36.259]
  MoveL 6119 to (7.04, 84.93, -279.16) mm, rotated rx -172.19 ry 6.28 rz 7.52 deg; joints [-8.792, -25.878, 75.637, 93.246, 106.286, 61.63, -36.259]
  MoveL 6120 to (6.79, 83.99, -279.63) mm, rotated rx -172.19 ry 6.28 rz 7.52 deg; joints [-8.792, -25.957, 75.746, 93.238, 106.287, 61.6, -36.259]
  MoveL 6121 to (6.32, 82.88, -279.91) mm, rotated rx -172.19 ry 6.28 rz 7.52 deg; joints [-8.782, -26.046, 75.879, 93.232, 106.283, 61.553, -36.259]
  MoveL 6122 to (5.61, 81.6, -280.01) mm, rotated rx -172.19 ry 6.28 rz 7.52 deg; joints [-8.764, -26.144, 76.037, 93.228, 106.275, 61.49, -36.259]
  MoveL 6123 to (5.34, 81.15, -280.01) mm, rotated rx -172.19 ry 6.28 rz 7.52 deg; joints [-8.757, -26.178, 76.093, 93.226, 106.272, 61.466, -36.259]
  MoveL 6124 to (5.09, 80.76, -279.99) mm, rotated rx -172.19 ry 6.28 rz 7.52 deg; joints [-8.75, -26.207, 76.143, 93.226, 106.268, 61.444, -36.259]
  MoveL 6125 to (4.86, 80.43, -279.94) mm, rotated rx -172.19 ry 6.28 rz 7.52 deg; joints [-8.743, -26.231, 76.186, 93.226, 106.265, 61.425, -36.259]
  MoveL 6126 to (4.64, 80.11, -279.88) mm, rotated rx -172.19 ry 6.28 rz 7.52 deg; joints [-8.736, -26.254, 76.227, 93.225, 106.262, 61.406, -36.259]
  MoveL 6127 to (4.4, 79.75, -279.84) mm, rotated rx -172.19 ry 6.28 rz 7.52 deg; joints [-8.729, -26.28, 76.272, 93.225, 106.258, 61.385, -36.259]
  MoveL 6128 to (4.13, 79.34, -279.82) mm, rotated rx -172.19 ry 6.28 rz 7.52 deg; joints [-8.722, -26.31, 76.324, 93.224, 106.255, 61.362, -36.259]
  MoveL 6129 to (3.86, 78.89, -279.82) mm, rotated rx -172.19 ry 6.28 rz 7.52 deg; joints [-8.714, -26.344, 76.38, 93.224, 106.251, 61.339, -36.259]
  MoveL 6130 to (3.62, 78.49, -279.8) mm, rotated rx -172.19 ry 6.28 rz 7.52 deg; joints [-8.707, -26.373, 76.43, 93.223, 106.248, 61.317, -36.259]
  MoveL 6131 to (3.4, 78.15, -279.74) mm, rotated rx -172.19 ry 6.28 rz 7.52 deg; joints [-8.701, -26.397, 76.473, 93.222, 106.245, 61.297, -36.259]
  MoveL 6132 to (3.18, 77.83, -279.68) mm, rotated rx -172.19 ry 6.28 rz 7.52 deg; joints [-8.694, -26.42, 76.515, 93.222, 106.241, 61.277, -36.259]
  MoveL 6133 to (2.94, 77.47, -279.64) mm, rotated rx -172.19 ry 6.28 rz 7.52 deg; joints [-8.687, -26.446, 76.561, 93.221, 106.238, 61.256, -36.259]
  MoveL 6134 to (2.68, 77.05, -279.61) mm, rotated rx -172.19 ry 6.28 rz 7.52 deg; joints [-8.68, -26.476, 76.613, 93.221, 106.235, 61.233, -36.259]
  MoveL 6135 to (2.41, 76.6, -279.61) mm, rotated rx -172.19 ry 6.28 rz 7.52 deg; joints [-8.672, -26.509, 76.668, 93.22, 106.231, 61.21, -36.259]
  MoveL 6136 to (1.84, 75.79, -279.59) mm, rotated rx -172.19 ry 6.28 rz 7.52 deg; joints [-8.656, -26.57, 76.769, 93.22, 106.223, 61.168, -36.259]
  MoveC 6137 to (1.02, 74.69, -279.59) mm, rotated rx -172.19 ry 6.28 rz 7.52 deg; joints [-8.633, -26.655, 76.906, 93.223, 106.211, 61.112, -36.259] to (0.33, 73.49, -279.59) mm, rotated rx -172.19 ry 6.28 rz 7.52 deg; joints [-8.614, -26.743, 77.054, 93.22, 106.203, 61.05, -36.259]
  MoveL 6138 to (0.33, 73.49, -279.58) mm, rotated rx -172.19 ry 6.28 rz 7.52 deg; joints [-8.614, -26.743, 77.054, 93.22, 106.203, 61.05, -36.259]
  MoveL 6139 to (-0.04, 72.95, -279.57) mm, rotated rx -172.19 ry 6.28 rz 7.52 deg; joints [-8.604, -26.784, 77.121, 93.22, 106.197, 61.021, -36.259]
  MoveL 6140 to (-0.41, 72.51, -279.54) mm, rotated rx -172.19 ry 6.28 rz 7.52 deg; joints [-8.593, -26.817, 77.176, 93.222, 106.192, 60.999, -36.259]
  MoveL 6141 to (-0.66, 72.33, -279.44) mm, rotated rx -172.19 ry 6.28 rz 7.52 deg; joints [-8.585, -26.829, 77.2, 93.225, 106.187, 60.986, -36.259]
  MoveL 6142 to (-0.65, 72.39, -279.24) mm, rotated rx -172.19 ry 6.28 rz 7.52 deg; joints [-8.582, -26.819, 77.196, 93.225, 106.186, 60.98, -36.259]
  MoveL 6143 to (-0.37, 72.71, -278.94) mm, rotated rx -172.19 ry 6.28 rz 7.52 deg; joints [-8.587, -26.785, 77.163, 93.221, 106.189, 60.98, -36.259]
  MoveL 6144 to (-0.47, 73.08, -278.31) mm, rotated rx -172.19 ry 6.28 rz 7.52 deg; joints [-8.577, -26.744, 77.129, 93.227, 106.183, 60.972, -36.259]
  MoveL 6145 to (-2.27, 72.12, -278.31) mm, rotated rx -172.19 ry 6.28 rz 7.52 deg; joints [-8.523, -26.833, 77.25, 93.258, 106.15, 60.936, -36.259]
  MoveL 6146 to (-4.2, 71.18, -278.25) mm, rotated rx -172.19 ry 6.28 rz 7.52 deg; joints [-8.464, -26.92, 77.369, 93.293, 106.115, 60.9, -36.259]
  MoveL 6147 to (-6.26, 70.23, -278.13) mm, rotated rx -172.19 ry 6.28 rz 7.52 deg; joints [-8.401, -27.008, 77.491, 93.332, 106.077, 60.862, -36.259]
  MoveL 6148 to (-8.29, 69.29, -278.03) mm, rotated rx -172.19 ry 6.28 rz 7.52 deg; joints [-8.339, -27.095, 77.611, 93.37, 106.039, 60.826, -36.259]
  MoveL 6149 to (-10.24, 68.39, -277.85) mm, rotated rx -172.19 ry 6.28 rz 7.52 deg; joints [-8.278, -27.176, 77.726, 93.407, 106.002, 60.788, -36.259]
  MoveL 6150 to (-12.01, 67.58, -277.71) mm, rotated rx -172.19 ry 6.28 rz 7.52 deg; joints [-8.223, -27.249, 77.829, 93.44, 105.969, 60.755, -36.259]
  MoveL 6151 to (-13.88, 66.7, -277.65) mm, rotated rx -172.19 ry 6.28 rz 7.52 deg; joints [-8.165, -27.331, 77.938, 93.476, 105.934, 60.724, -36.259]
  MoveL 6152 to (-15.84, 65.79, -277.58) mm, rotated rx -172.19 ry 6.28 rz 7.52 deg; joints [-8.105, -27.415, 78.052, 93.513, 105.898, 60.692, -36.259]
  MoveL 6153 to (-17.97, 64.8, -277.43) mm, rotated rx -172.19 ry 6.28 rz 7.52 deg; joints [-8.039, -27.505, 78.176, 93.554, 105.858, 60.652, -36.259]
  MoveL 6154 to (-19.67, 64, -277.32) mm, rotated rx -172.19 ry 6.28 rz 7.52 deg; joints [-7.986, -27.576, 78.276, 93.586, 105.827, 60.622, -36.259]
  MoveL 6155 to (-21.83, 62.99, -277.1) mm, rotated rx -172.19 ry 6.28 rz 7.52 deg; joints [-7.918, -27.665, 78.403, 93.627, 105.786, 60.579, -36.259]
  MoveL 6156 to (-23.53, 62.19, -276.99) mm, rotated rx -172.19 ry 6.28 rz 7.52 deg; joints [-7.865, -27.737, 78.502, 93.66, 105.754, 60.549, -36.259]
  MoveL 6157 to (-25.46, 61.27, -276.82) mm, rotated rx -172.19 ry 6.28 rz 7.52 deg; joints [-7.805, -27.818, 78.615, 93.697, 105.718, 60.512, -36.259]
  MoveL 6158 to (-27.62, 60.25, -276.77) mm, rotated rx -172.19 ry 6.28 rz 7.52 deg; joints [-7.738, -27.911, 78.739, 93.739, 105.679, 60.478, -36.259]
  MoveL 6159 to (-29.32, 59.45, -276.66) mm, rotated rx -172.19 ry 6.28 rz 7.52 deg; joints [-7.685, -27.983, 78.837, 93.772, 105.647, 60.448, -36.259]
  MoveL 6160 to (-31.24, 58.52, -276.5) mm, rotated rx -172.19 ry 6.28 rz 7.52 deg; joints [-7.625, -28.063, 78.95, 93.809, 105.611, 60.412, -36.259]
  MoveL 6161 to (-33.4, 57.5, -276.45) mm, rotated rx -172.19 ry 6.28 rz 7.52 deg; joints [-7.558, -28.157, 79.072, 93.852, 105.571, 60.379, -36.259]
  MoveL 6162 to (-35.1, 56.69, -276.34) mm, rotated rx -172.19 ry 6.28 rz 7.52 deg; joints [-7.505, -28.228, 79.171, 93.885, 105.539, 60.349, -36.259]
  MoveL 6163 to (-37.1, 55.73, -276.23) mm, rotated rx -172.19 ry 6.28 rz 7.52 deg; joints [-7.443, -28.313, 79.286, 93.925, 105.502, 60.315, -36.259]
  MoveL 6164 to (-39.11, 54.77, -276.17) mm, rotated rx -172.19 ry 6.28 rz 7.52 deg; joints [-7.381, -28.4, 79.4, 93.965, 105.465, 60.284, -36.259]
  MoveL 6165 to (-40.79, 53.93, -275.99) mm, rotated rx -172.19 ry 6.28 rz 7.52 deg; joints [-7.327, -28.47, 79.501, 93.997, 105.434, 60.25, -36.259]
  MoveL 6166 to (-42.33, 53.13, -275.73) mm, rotated rx -172.19 ry 6.28 rz 7.52 deg; joints [-7.277, -28.534, 79.599, 94.026, 105.405, 60.212, -36.259]
  MoveL 6167 to (-43.76, 52.36, -275.38) mm, rotated rx -172.19 ry 6.28 rz 7.52 deg; joints [-7.23, -28.592, 79.696, 94.052, 105.378, 60.17, -36.259]
  MoveL 6168 to (-42.27, 52.6, -274.69) mm, rotated rx -172.19 ry 6.28 rz 7.52 deg; joints [-7.269, -28.537, 79.681, 94.011, 105.405, 60.129, -36.259]
  MoveL 6169 to (-42.49, 52.54, -274.69) mm, rotated rx -172.19 ry 6.28 rz 7.52 deg; joints [-7.262, -28.543, 79.688, 94.016, 105.401, 60.129, -36.259]
  MoveL 6170 to (-42.79, 52.5, -274.67) mm, rotated rx -172.19 ry 6.28 rz 7.52 deg; joints [-7.252, -28.549, 79.692, 94.024, 105.395, 60.13, -36.259]
  MoveL 6171 to (-43.24, 52.51, -274.64) mm, rotated rx -172.19 ry 6.28 rz 7.52 deg; joints [-7.238, -28.553, 79.691, 94.036, 105.385, 60.135, -36.259]
  MoveL 6172 to (-43.78, 52.55, -274.6) mm, rotated rx -172.19 ry 6.28 rz 7.52 deg; joints [-7.22, -28.557, 79.687, 94.052, 105.374, 60.142, -36.259]
  MoveL 6173 to (-44.39, 52.62, -274.56) mm, rotated rx -172.19 ry 6.28 rz 7.52 deg; joints [-7.2, -28.559, 79.679, 94.07, 105.361, 60.151, -36.259]
  MoveL 6174 to (-46.98, 53.01, -274.56) mm, rotated rx -172.19 ry 6.28 rz 7.52 deg; joints [-7.119, -28.568, 79.631, 94.148, 105.305, 60.207, -36.259]
  MoveL 6175 to (-47.59, 53.08, -274.53) mm, rotated rx -172.19 ry 6.28 rz 7.52 deg; joints [-7.099, -28.57, 79.622, 94.166, 105.292, 60.217, -36.259]
  MoveL 6176 to (-48.27, 53.16, -274.47) mm, rotated rx -172.19 ry 6.28 rz 7.52 deg; joints [-7.077, -28.572, 79.613, 94.186, 105.278, 60.227, -36.259]
  MoveL 6177 to (-48.89, 53.23, -274.44) mm, rotated rx -172.19 ry 6.28 rz 7.52 deg; joints [-7.057, -28.574, 79.604, 94.204, 105.264, 60.238, -36.259]
  MoveL 6178 to (-49.41, 53.31, -274.44) mm, rotated rx -172.19 ry 6.28 rz 7.52 deg; joints [-7.041, -28.576, 79.594, 94.22, 105.253, 60.249, -36.259]
  MoveL 6179 to (-49.89, 53.38, -274.43) mm, rotated rx -172.19 ry 6.28 rz 7.52 deg; joints [-7.025, -28.577, 79.585, 94.234, 105.243, 60.259, -36.259]
  MoveL 6180 to (-50.41, 53.46, -274.43) mm, rotated rx -172.19 ry 6.28 rz 7.52 deg; joints [-7.009, -28.579, 79.575, 94.25, 105.231, 60.27, -36.259]
  MoveL 6181 to (-50.92, 53.54, -274.43) mm, rotated rx -172.19 ry 6.28 rz 7.52 deg; joints [-6.993, -28.58, 79.566, 94.265, 105.221, 60.281, -36.259]
  MoveL 6182 to (-51.4, 53.6, -274.4) mm, rotated rx -172.19 ry 6.28 rz 7.52 deg; joints [-6.977, -28.582, 79.558, 94.28, 105.21, 60.289, -36.259]
  MoveL 6183 to (-51.86, 53.65, -274.36) mm, rotated rx -172.19 ry 6.28 rz 7.52 deg; joints [-6.962, -28.583, 79.553, 94.293, 105.2, 60.296, -36.259]
  MoveL 6184 to (-52.35, 53.72, -274.34) mm, rotated rx -172.19 ry 6.28 rz 7.52 deg; joints [-6.946, -28.584, 79.545, 94.308, 105.19, 60.305, -36.259]
  MoveL 6185 to (-52.88, 53.8, -274.33) mm, rotated rx -172.19 ry 6.28 rz 7.52 deg; joints [-6.93, -28.586, 79.535, 94.323, 105.178, 60.316, -36.259]
  MoveL 6186 to (-53.92, 53.95, -274.33) mm, rotated rx -172.19 ry 6.28 rz 7.52 deg; joints [-6.897, -28.589, 79.514, 94.355, 105.156, 60.338, -36.259]
  Set speed (1000.0 mm/s)
  MoveL 6187 to (-73.51, 63.09, -274.33) mm, rotated rx -172.19 ry 6.28 rz 7.52 deg; joints [-6.274, -28.239, 78.384, 95.034, 104.697, 61.11, -36.259]
  Print: /'Flow1'
  Set speed (1000.0 mm/s)
  MoveL 6188 to (-38.6, -107.51, -82.29) mm, rotated rx 81.04 ry 30.21 rz 20.91 deg; joints [-3.376, -17.615, 78.362, 104.464, 105.536, 55.041, -153.967]
  Set speed (1000.0 mm/s)
  MoveL 6189 to (-1.84, -81.77, -82.29) mm, rotated rx 81.04 ry 30.21 rz 20.91 deg; joints [-4.553, -18.227, 81.087, 102.873, 106.576, 53.042, -153.967]
  Set speed (100.0 mm/s)
  MoveL 6190 to (57.77, -40.03, -82.29) mm, rotated rx 81.04 ry 30.21 rz 20.91 deg; joints [-6.543, -18.987, 85.101, 100.135, 108.065, 49.881, -153.967]
  MoveL 6191 to (58.29, -40.06, -82.29) mm, rotated rx 81.04 ry 30.21 rz 20.91 deg; joints [-6.56, -18.999, 85.117, 100.119, 108.073, 49.879, -153.967]
  MoveL 6192 to (58.93, -40.04, -82.19) mm, rotated rx 81.04 ry 30.21 rz 20.91 deg; joints [-6.581, -19.02, 85.147, 100.097, 108.083, 49.87, -153.967]
  MoveL 6193 to (59.52, -40.04, -82.13) mm, rotated rx 81.04 ry 30.21 rz 20.91 deg; joints [-6.6, -19.036, 85.171, 100.078, 108.092, 49.863, -153.967]
  MoveL 6194 to (60.09, -40.06, -82.11) mm, rotated rx 81.04 ry 30.21 rz 20.91 deg; joints [-6.619, -19.051, 85.19, 100.059, 108.1, 49.86, -153.967]
  MoveL 6195 to (63.75, -40.26, -82.11) mm, rotated rx 81.04 ry 30.21 rz 20.91 deg; joints [-6.741, -19.136, 85.297, 99.943, 108.153, 49.847, -153.967]
  MoveL 6196 to (65.2, -40.4, -82.2) mm, rotated rx 81.04 ry 30.21 rz 20.91 deg; joints [-6.791, -19.165, 85.327, 99.899, 108.172, 49.849, -153.967]
  MoveL 6197 to (66.36, -40.64, -82.47) mm, rotated rx 81.04 ry 30.21 rz 20.91 deg; joints [-6.832, -19.178, 85.326, 99.866, 108.187, 49.866, -153.967]
  MoveL 6198 to (67.24, -40.99, -82.91) mm, rotated rx 81.04 ry 30.21 rz 20.91 deg; joints [-6.866, -19.175, 85.295, 99.845, 108.195, 49.898, -153.967]
  MoveL 6199 to (67.57, -41.21, -83.2) mm, rotated rx 81.04 ry 30.21 rz 20.91 deg; joints [-6.881, -19.168, 85.268, 99.839, 108.198, 49.92, -153.967]
  MoveL 6200 to (67.83, -41.45, -83.53) mm, rotated rx 81.04 ry 30.21 rz 20.91 deg; joints [-6.893, -19.156, 85.232, 99.836, 108.198, 49.946, -153.967]
  MoveL 6201 to (68.15, -42.01, -84.33) mm, rotated rx 81.04 ry 30.21 rz 20.91 deg; joints [-6.912, -19.122, 85.139, 99.838, 108.196, 50.008, -153.967]
  MoveL 6202 to (68.18, -42.68, -85.31) mm, rotated rx 81.04 ry 30.21 rz 20.91 deg; joints [-6.923, -19.071, 85.015, 99.852, 108.188, 50.086, -153.967]
  MoveL 6203 to (67.4, -44.34, -87.79) mm, rotated rx 81.04 ry 30.21 rz 20.91 deg; joints [-6.923, -18.922, 84.673, 99.914, 108.155, 50.286, -153.967]
  MoveL 6204 to (65.83, -45.9, -90.28) mm, rotated rx 81.04 ry 30.21 rz 20.91 deg; joints [-6.896, -18.754, 84.308, 100.001, 108.11, 50.487, -153.967]
  MoveL 6205 to (63.82, -46.87, -92.05) mm, rotated rx 81.04 ry 30.21 rz 20.91 deg; joints [-6.848, -18.61, 84.026, 100.088, 108.066, 50.627, -153.967]
  MoveL 6206 to (62.64, -47.12, -92.67) mm, rotated rx 81.04 ry 30.21 rz 20.91 deg; joints [-6.816, -18.548, 83.916, 100.132, 108.044, 50.674, -153.967]
  MoveL 6207 to (61.36, -47.23, -93.12) mm, rotated rx 81.04 ry 30.21 rz 20.91 deg; joints [-6.778, -18.492, 83.826, 100.177, 108.023, 50.706, -153.967]
  MoveL 6208 to (58.45, -47, -93.47) mm, rotated rx 81.04 ry 30.21 rz 20.91 deg; joints [-6.685, -18.4, 83.709, 100.266, 107.98, 50.725, -153.967]
  MoveL 6209 to (55.35, -46.47, -93.48) mm, rotated rx 81.04 ry 30.21 rz 20.91 deg; joints [-6.583, -18.321, 83.633, 100.356, 107.939, 50.714, -153.967]
  MoveL 6210 to (54.86, -46.4, -93.5) mm, rotated rx 81.04 ry 30.21 rz 20.91 deg; joints [-6.567, -18.308, 83.619, 100.37, 107.932, 50.714, -153.967]
  MoveL 6211 to (54.41, -46.35, -93.54) mm, rotated rx 81.04 ry 30.21 rz 20.91 deg; joints [-6.552, -18.294, 83.603, 100.384, 107.926, 50.715, -153.967]
  MoveL 6212 to (53.99, -46.32, -93.6) mm, rotated rx 81.04 ry 30.21 rz 20.91 deg; joints [-6.539, -18.28, 83.585, 100.397, 107.92, 50.718, -153.967]
  MoveL 6213 to (53.55, -46.27, -93.65) mm, rotated rx 81.04 ry 30.21 rz 20.91 deg; joints [-6.525, -18.267, 83.567, 100.411, 107.913, 50.721, -153.967]
  MoveL 6214 to (53.01, -46.2, -93.67) mm, rotated rx 81.04 ry 30.21 rz 20.91 deg; joints [-6.508, -18.251, 83.551, 100.427, 107.906, 50.721, -153.967]
  MoveL 6215 to (52.36, -46.11, -93.71) mm, rotated rx 81.04 ry 30.21 rz 20.91 deg; joints [-6.487, -18.233, 83.53, 100.446, 107.897, 50.721, -153.967]
  MoveL 6216 to (51.81, -46.05, -93.77) mm, rotated rx 81.04 ry 30.21 rz 20.91 deg; joints [-6.469, -18.216, 83.509, 100.463, 107.889, 50.724, -153.967]
  MoveL 6217 to (51.36, -46.02, -93.84) mm, rotated rx 81.04 ry 30.21 rz 20.91 deg; joints [-6.455, -18.2, 83.489, 100.477, 107.882, 50.728, -153.967]
  MoveL 6218 to (50.93, -45.97, -93.89) mm, rotated rx 81.04 ry 30.21 rz 20.91 deg; joints [-6.441, -18.186, 83.472, 100.49, 107.876, 50.73, -153.967]
  MoveL 6219 to (50.45, -45.9, -93.91) mm, rotated rx 81.04 ry 30.21 rz 20.91 deg; joints [-6.426, -18.173, 83.457, 100.504, 107.869, 50.73, -153.967]
  MoveL 6220 to (49.94, -45.82, -93.91) mm, rotated rx 81.04 ry 30.21 rz 20.91 deg; joints [-6.409, -18.16, 83.445, 100.519, 107.862, 50.728, -153.967]
  MoveL 6221 to (49.4, -45.73, -93.92) mm, rotated rx 81.04 ry 30.21 rz 20.91 deg; joints [-6.391, -18.146, 83.431, 100.534, 107.855, 50.726, -153.967]
  MoveL 6222 to (48.84, -45.64, -93.93) mm, rotated rx 81.04 ry 30.21 rz 20.91 deg; joints [-6.373, -18.131, 83.415, 100.551, 107.847, 50.726, -153.967]
  MoveL 6223 to (48.18, -45.57, -93.96) mm, rotated rx 81.04 ry 30.21 rz 20.91 deg; joints [-6.352, -18.113, 83.394, 100.57, 107.838, 50.727, -153.967]
  MoveL 6224 to (47.59, -45.53, -94.03) mm, rotated rx 81.04 ry 30.21 rz 20.91 deg; joints [-6.333, -18.095, 83.37, 100.589, 107.829, 50.732, -153.967]
  MoveL 6225 to (47.14, -45.53, -94.13) mm, rotated rx 81.04 ry 30.21 rz 20.91 deg; joints [-6.319, -18.078, 83.345, 100.604, 107.822, 50.739, -153.967]
  MoveL 6226 to (47.14, -45.52, -94.37) mm, rotated rx 81.04 ry 30.21 rz 20.91 deg; joints [-6.322, -18.062, 83.322, 100.604, 107.822, 50.747, -153.967]
  MoveL 6227 to (47.53, -45.46, -94.72) mm, rotated rx 81.04 ry 30.21 rz 20.91 deg; joints [-6.339, -18.047, 83.302, 100.59, 107.828, 50.753, -153.967]
  MoveL 6228 to (48.14, -46.05, -95.69) mm, rotated rx 81.04 ry 30.21 rz 20.91 deg; joints [-6.369, -18.008, 83.2, 100.583, 107.829, 50.821, -153.967]
  MoveL 6229 to (46.19, -46.92, -95.69) mm, rotated rx 81.04 ry 30.21 rz 20.91 deg; joints [-6.304, -17.978, 83.095, 100.664, 107.788, 50.892, -153.967]
  MoveL 6230 to (44.11, -47.89, -95.82) mm, rotated rx 81.04 ry 30.21 rz 20.91 deg; joints [-6.236, -17.937, 82.969, 100.751, 107.744, 50.975, -153.967]
  MoveL 6231 to (42.13, -48.79, -95.87) mm, rotated rx 81.04 ry 30.21 rz 20.91 deg; joints [-6.17, -17.902, 82.856, 100.834, 107.702, 51.051, -153.967]
  MoveL 6232 to (40.2, -49.67, -96) mm, rotated rx 81.04 ry 30.21 rz 20.91 deg; joints [-6.107, -17.863, 82.737, 100.914, 107.661, 51.128, -153.967]
  MoveL 6233 to (38.26, -50.57, -96.16) mm, rotated rx 81.04 ry 30.21 rz 20.91 deg; joints [-6.044, -17.822, 82.614, 100.995, 107.619, 51.206, -153.967]
  MoveL 6234 to (36.32, -51.45, -96.28) mm, rotated rx 81.04 ry 30.21 rz 20.91 deg; joints [-5.981, -17.783, 82.496, 101.075, 107.577, 51.283, -153.967]
  MoveL 6235 to (34.38, -52.35, -96.49) mm, rotated rx 81.04 ry 30.21 rz 20.91 deg; joints [-5.918, -17.739, 82.367, 101.156, 107.535, 51.363, -153.967]
  MoveL 6236 to (32.44, -53.22, -96.61) mm, rotated rx 81.04 ry 30.21 rz 20.91 deg; joints [-5.855, -17.7, 82.249, 101.236, 107.493, 51.44, -153.967]
  MoveL 6237 to (30.48, -54.1, -96.66) mm, rotated rx 81.04 ry 30.21 rz 20.91 deg; joints [-5.791, -17.664, 82.135, 101.317, 107.451, 51.514, -153.967]
  MoveL 6238 to (28.52, -54.99, -96.81) mm, rotated rx 81.04 ry 30.21 rz 20.91 deg; joints [-5.727, -17.622, 82.011, 101.397, 107.408, 51.593, -153.967]
  MoveL 6239 to (26.49, -55.9, -96.99) mm, rotated rx 81.04 ry 30.21 rz 20.91 deg; joints [-5.662, -17.576, 81.88, 101.481, 107.363, 51.675, -153.967]
  MoveL 6240 to (24.45, -56.81, -97.17) mm, rotated rx 81.04 ry 30.21 rz 20.91 deg; joints [-5.597, -17.53, 81.748, 101.564, 107.318, 51.757, -153.967]
  MoveL 6241 to (22.74, -57.57, -97.41) mm, rotated rx 81.04 ry 30.21 rz 20.91 deg; joints [-5.543, -17.485, 81.628, 101.634, 107.28, 51.829, -153.967]
  MoveL 6242 to (20.3, -58.66, -97.52) mm, rotated rx 81.04 ry 30.21 rz 20.91 deg; joints [-5.464, -17.437, 81.481, 101.733, 107.226, 51.923, -153.967]
  Set speed (1000.0 mm/s)
  MoveL 6243 to (-16.81, -84.64, -97.52) mm, rotated rx 81.04 ry 30.21 rz 20.91 deg; joints [-4.254, -16.887, 78.844, 103.388, 106.236, 53.925, -153.967]
  Set speed (1000.0 mm/s)
  MoveL 6244 to (-20.1, -79.94, -109.4) mm, rotated rx 81.04 ry 30.21 rz 20.91 deg; joints [-4.292, -15.95, 77.727, 103.406, 106.212, 54.112, -153.967]
  Set speed (100.0 mm/s)
  MoveL 6245 to (3.4, -63.49, -109.4) mm, rotated rx 81.04 ry 30.21 rz 20.91 deg; joints [-5.052, -16.318, 79.433, 102.369, 106.853, 52.833, -153.967]
  MoveL 6246 to (5.05, -63.01, -109.15) mm, rotated rx 81.04 ry 30.21 rz 20.91 deg; joints [-5.102, -16.368, 79.542, 102.308, 106.888, 52.778, -153.967]
  MoveL 6247 to (6.98, -62.41, -109.09) mm, rotated rx 81.04 ry 30.21 rz 20.91 deg; joints [-5.164, -16.411, 79.648, 102.235, 106.929, 52.719, -153.967]
  MoveL 6248 to (8.95, -61.81, -108.94) mm, rotated rx 81.04 ry 30.21 rz 20.91 deg; joints [-5.227, -16.459, 79.764, 102.162, 106.97, 52.657, -153.967]
  MoveL 6249 to (11.3, -61.1, -108.81) mm, rotated rx 81.04 ry 30.21 rz 20.91 deg; joints [-5.302, -16.515, 79.897, 102.073, 107.019, 52.585, -153.967]
  MoveL 6250 to (13.34, -60.47, -108.81) mm, rotated rx 81.04 ry 30.21 rz 20.91 deg; joints [-5.368, -16.555, 80.001, 101.997, 107.062, 52.526, -153.967]
  MoveL 6251 to (15.59, -59.76, -108.65) mm, rotated rx 81.04 ry 30.21 rz 20.91 deg; joints [-5.44, -16.609, 80.132, 101.911, 107.109, 52.455, -153.967]
  MoveL 6252 to (17.5, -59.18, -108.47) mm, rotated rx 81.04 ry 30.21 rz 20.91 deg; joints [-5.5, -16.659, 80.247, 101.84, 107.149, 52.394, -153.967]
  MoveL 6253 to (19.45, -58.58, -108.37) mm, rotated rx 81.04 ry 30.21 rz 20.91 deg; joints [-5.563, -16.703, 80.355, 101.766, 107.189, 52.334, -153.967]
  MoveL 6254 to (21.49, -57.94, -108.16) mm, rotated rx 81.04 ry 30.21 rz 20.91 deg; joints [-5.627, -16.756, 80.48, 101.688, 107.231, 52.267, -153.967]
  MoveL 6255 to (23.51, -57.3, -108) mm, rotated rx 81.04 ry 30.21 rz 20.91 deg; joints [-5.692, -16.805, 80.597, 101.612, 107.273, 52.203, -153.967]
  MoveL 6256 to (25.52, -56.67, -107.89) mm, rotated rx 81.04 ry 30.21 rz 20.91 deg; joints [-5.756, -16.851, 80.709, 101.535, 107.315, 52.141, -153.967]
  MoveL 6257 to (27.56, -56.02, -107.72) mm, rotated rx 81.04 ry 30.21 rz 20.91 deg; joints [-5.822, -16.901, 80.828, 101.457, 107.357, 52.075, -153.967]
  MoveL 6258 to (29.58, -55.37, -107.58) mm, rotated rx 81.04 ry 30.21 rz 20.91 deg; joints [-5.887, -16.948, 80.944, 101.379, 107.398, 52.011, -153.967]
  MoveL 6259 to (31.66, -54.71, -107.51) mm, rotated rx 81.04 ry 30.21 rz 20.91 deg; joints [-5.954, -16.991, 81.053, 101.3, 107.44, 51.95, -153.967]
  MoveL 6260 to (33.69, -54.05, -107.3) mm, rotated rx 81.04 ry 30.21 rz 20.91 deg; joints [-6.019, -17.043, 81.176, 101.222, 107.482, 51.882, -153.967]
  MoveL 6261 to (35.71, -53.4, -107.18) mm, rotated rx 81.04 ry 30.21 rz 20.91 deg; joints [-6.084, -17.088, 81.288, 101.144, 107.522, 51.819, -153.967]
  MoveL 6262 to (37.76, -52.73, -107.06) mm, rotated rx 81.04 ry 30.21 rz 20.91 deg; joints [-6.151, -17.134, 81.402, 101.065, 107.564, 51.755, -153.967]
  MoveL 6263 to (39.41, -52.06, -106.85) mm, rotated rx 81.04 ry 30.21 rz 20.91 deg; joints [-6.203, -17.175, 81.51, 100.998, 107.599, 51.691, -153.967]
  MoveL 6264 to (40.71, -51.38, -106.5) mm, rotated rx 81.04 ry 30.21 rz 20.91 deg; joints [-6.242, -17.218, 81.622, 100.942, 107.629, 51.624, -153.967]
  MoveL 6265 to (41.68, -50.66, -105.97) mm, rotated rx 81.04 ry 30.21 rz 20.91 deg; joints [-6.269, -17.264, 81.741, 100.896, 107.654, 51.55, -153.967]
  MoveL 6266 to (40.15, -50.66, -105.11) mm, rotated rx 81.04 ry 30.21 rz 20.91 deg; joints [-6.209, -17.285, 81.776, 100.944, 107.631, 51.53, -153.967]
  MoveL 6267 to (40.94, -50.59, -105.11) mm, rotated rx 81.04 ry 30.21 rz 20.91 deg; joints [-6.235, -17.302, 81.806, 100.917, 107.645, 51.519, -153.967]
  MoveL 6268 to (41.65, -50.59, -105.11) mm, rotated rx 81.04 ry 30.21 rz 20.91 deg; joints [-6.258, -17.318, 81.83, 100.895, 107.656, 51.513, -153.967]
  MoveL 6269 to (42.28, -50.69, -105.11) mm, rotated rx 81.04 ry 30.21 rz 20.91 deg; joints [-6.279, -17.335, 81.847, 100.876, 107.665, 51.514, -153.967]
  MoveL 6270 to (42.93, -50.83, -105.09) mm, rotated rx 81.04 ry 30.21 rz 20.91 deg; joints [-6.3, -17.353, 81.864, 100.858, 107.673, 51.518, -153.967]
  MoveL 6271 to (43.67, -51.02, -105.05) mm, rotated rx 81.04 ry 30.21 rz 20.91 deg; joints [-6.324, -17.375, 81.883, 100.838, 107.683, 51.522, -153.967]
  MoveL 6272 to (45.68, -51.62, -105.05) mm, rotated rx 81.04 ry 30.21 rz 20.91 deg; joints [-6.389, -17.431, 81.922, 100.786, 107.708, 51.545, -153.967]
  MoveL 6273 to (46.11, -51.73, -105.03) mm, rotated rx 81.04 ry 30.21 rz 20.91 deg; joints [-6.403, -17.444, 81.933, 100.775, 107.713, 51.548, -153.967]
  MoveL 6274 to (47.11, -52.03, -105.03) mm, rotated rx 81.04 ry 30.21 rz 20.91 deg; joints [-6.436, -17.471, 81.953, 100.748, 107.725, 51.56, -153.967]
  MoveL 6275 to (47.6, -52.17, -105.03) mm, rotated rx 81.04 ry 30.21 rz 20.91 deg; joints [-6.451, -17.485, 81.963, 100.736, 107.731, 51.565, -153.967]
  MoveL 6276 to (48.07, -52.3, -105.01) mm, rotated rx 81.04 ry 30.21 rz 20.91 deg; joints [-6.467, -17.499, 81.974, 100.723, 107.737, 51.569, -153.967]
  MoveL 6277 to (48.53, -52.41, -104.98) mm, rotated rx 81.04 ry 30.21 rz 20.91 deg; joints [-6.481, -17.514, 81.988, 100.711, 107.743, 51.571, -153.967]
  MoveL 6278 to (48.96, -52.5, -104.92) mm, rotated rx 81.04 ry 30.21 rz 20.91 deg; joints [-6.495, -17.528, 82.003, 100.699, 107.749, 51.571, -153.967]
  MoveL 6279 to (49.42, -52.61, -104.88) mm, rotated rx 81.04 ry 30.21 rz 20.91 deg; joints [-6.509, -17.543, 82.017, 100.686, 107.755, 51.573, -153.967]
  MoveL 6280 to (49.9, -52.74, -104.86) mm, rotated rx 81.04 ry 30.21 rz 20.91 deg; joints [-6.525, -17.557, 82.028, 100.674, 107.761, 51.577, -153.967]
  MoveL 6281 to (50.39, -52.88, -104.86) mm, rotated rx 81.04 ry 30.21 rz 20.91 deg; joints [-6.541, -17.571, 82.039, 100.661, 107.767, 51.582, -153.967]
  MoveL 6282 to (50.86, -53.01, -104.84) mm, rotated rx 81.04 ry 30.21 rz 20.91 deg; joints [-6.556, -17.585, 82.05, 100.648, 107.773, 51.586, -153.967]
  MoveL 6283 to (51.33, -53.12, -104.8) mm, rotated rx 81.04 ry 30.21 rz 20.91 deg; joints [-6.571, -17.6, 82.064, 100.635, 107.779, 51.588, -153.967]
  MoveL 6284 to (51.75, -53.2, -104.75) mm, rotated rx 81.04 ry 30.21 rz 20.91 deg; joints [-6.584, -17.614, 82.08, 100.623, 107.785, 51.588, -153.967]
  MoveL 6285 to (52.2, -53.28, -104.69) mm, rotated rx 81.04 ry 30.21 rz 20.91 deg; joints [-6.598, -17.629, 82.096, 100.611, 107.791, 51.588, -153.967]
  MoveL 6286 to (53.6, -53.63, -104.61) mm, rotated rx 81.04 ry 30.21 rz 20.91 deg; joints [-6.643, -17.672, 82.134, 100.573, 107.809, 51.597, -153.967]
  MoveL 6287 to (54.7, -54.05, -104.74) mm, rotated rx 81.04 ry 30.21 rz 20.91 deg; joints [-6.68, -17.695, 82.137, 100.547, 107.822, 51.621, -153.967]
  MoveL 6288 to (55.5, -54.55, -105.07) mm, rotated rx 81.04 ry 30.21 rz 20.91 deg; joints [-6.71, -17.699, 82.106, 100.532, 107.828, 51.659, -153.967]
  MoveL 6289 to (55.79, -54.83, -105.32) mm, rotated rx 81.04 ry 30.21 rz 20.91 deg; joints [-6.722, -17.694, 82.077, 100.529, 107.829, 51.684, -153.967]
  MoveL 6290 to (56, -55.13, -105.62) mm, rotated rx 81.04 ry 30.21 rz 20.91 deg; joints [-6.732, -17.683, 82.04, 100.528, 107.828, 51.713, -153.967]
  MoveL 6291 to (56.21, -55.78, -106.38) mm, rotated rx 81.04 ry 30.21 rz 20.91 deg; joints [-6.746, -17.648, 81.939, 100.536, 107.822, 51.782, -153.967]
  MoveL 6292 to (56.11, -56.51, -107.35) mm, rotated rx 81.04 ry 30.21 rz 20.91 deg; joints [-6.753, -17.594, 81.804, 100.556, 107.81, 51.866, -153.967]
  MoveL 6293 to (55.03, -58.21, -109.91) mm, rotated rx 81.04 ry 30.21 rz 20.91 deg; joints [-6.744, -17.426, 81.428, 100.629, 107.768, 52.08, -153.967]
  MoveL 6294 to (53.2, -59.67, -112.52) mm, rotated rx 81.04 ry 30.21 rz 20.91 deg; joints [-6.711, -17.234, 81.033, 100.722, 107.716, 52.287, -153.967]
  MoveL 6295 to (52.17, -60.11, -113.55) mm, rotated rx 81.04 ry 30.21 rz 20.91 deg; joints [-6.688, -17.149, 80.873, 100.765, 107.693, 52.362, -153.967]
  MoveL 6296 to (51.06, -60.35, -114.39) mm, rotated rx 81.04 ry 30.21 rz 20.91 deg; joints [-6.661, -17.072, 80.739, 100.807, 107.67, 52.418, -153.967]
  MoveL 6297 to (49.87, -60.4, -115.04) mm, rotated rx 81.04 ry 30.21 rz 20.91 deg; joints [-6.63, -17.002, 80.631, 100.846, 107.649, 52.455, -153.967]
  MoveL 6298 to (48.61, -60.26, -115.51) mm, rotated rx 81.04 ry 30.21 rz 20.91 deg; joints [-6.594, -16.94, 80.548, 100.884, 107.629, 52.473, -153.967]
  MoveL 6299 to (47.27, -59.91, -115.79) mm, rotated rx 81.04 ry 30.21 rz 20.91 deg; joints [-6.553, -16.885, 80.491, 100.92, 107.611, 52.473, -153.967]
  MoveL 6300 to (45.85, -59.38, -115.88) mm, rotated rx 81.04 ry 30.21 rz 20.91 deg; joints [-6.509, -16.839, 80.459, 100.954, 107.595, 52.453, -153.967]
  MoveL 6301 to (42.95, -58.12, -115.88) mm, rotated rx 81.04 ry 30.21 rz 20.91 deg; joints [-6.415, -16.753, 80.422, 101.02, 107.563, 52.395, -153.967]
  MoveL 6302 to (42.44, -57.9, -115.9) mm, rotated rx 81.04 ry 30.21 rz 20.91 deg; joints [-6.399, -16.737, 80.413, 101.032, 107.557, 52.386, -153.967]
  MoveL 6303 to (41.86, -57.68, -115.93) mm, rotated rx 81.04 ry 30.21 rz 20.91 deg; joints [-6.381, -16.718, 80.401, 101.046, 107.551, 52.378, -153.967]
  MoveL 6304 to (41.14, -57.43, -116.03) mm, rotated rx 81.04 ry 30.21 rz 20.91 deg; joints [-6.359, -16.692, 80.378, 101.064, 107.542, 52.371, -153.967]
  MoveL 6305 to (40.57, -57.21, -116.06) mm, rotated rx 81.04 ry 30.21 rz 20.91 deg; joints [-6.34, -16.672, 80.366, 101.078, 107.535, 52.363, -153.967]
  MoveL 6306 to (40.06, -57, -116.08) mm, rotated rx 81.04 ry 30.21 rz 20.91 deg; joints [-6.324, -16.657, 80.357, 101.089, 107.53, 52.354, -153.967]
  MoveL 6307 to (39.6, -56.8, -116.09) mm, rotated rx 81.04 ry 30.21 rz 20.91 deg; joints [-6.309, -16.642, 80.35, 101.1, 107.524, 52.346, -153.967]
  MoveL 6308 to (39.17, -56.63, -116.1) mm, rotated rx 81.04 ry 30.21 rz 20.91 deg; joints [-6.296, -16.629, 80.342, 101.11, 107.52, 52.339, -153.967]
  MoveL 6309 to (37.28, -55.82, -116.11) mm, rotated rx 81.04 ry 30.21 rz 20.91 deg; joints [-6.235, -16.573, 80.315, 101.154, 107.499, 52.303, -153.967]
  MoveL 6310 to (36.8, -55.63, -116.15) mm, rotated rx 81.04 ry 30.21 rz 20.91 deg; joints [-6.22, -16.556, 80.304, 101.165, 107.494, 52.296, -153.967]
  MoveL 6311 to (36.36, -55.48, -116.2) mm, rotated rx 81.04 ry 30.21 rz 20.91 deg; joints [-6.206, -16.54, 80.291, 101.177, 107.488, 52.292, -153.967]
  MoveL 6312 to (35.92, -55.35, -116.27) mm, rotated rx 81.04 ry 30.21 rz 20.91 deg; joints [-6.193, -16.523, 80.275, 101.188, 107.482, 52.29, -153.967]
  MoveL 6313 to (35.44, -55.23, -116.33) mm, rotated rx 81.04 ry 30.21 rz 20.91 deg; joints [-6.178, -16.506, 80.258, 101.201, 107.476, 52.289, -153.967]
  MoveL 6314 to (34.9, -55.11, -116.36) mm, rotated rx 81.04 ry 30.21 rz 20.91 deg; joints [-6.161, -16.49, 80.242, 101.216, 107.469, 52.287, -153.967]
  MoveL 6315 to (34.23, -55.06, -116.37) mm, rotated rx 81.04 ry 30.21 rz 20.91 deg; joints [-6.139, -16.473, 80.22, 101.236, 107.458, 52.29, -153.967]
  MoveL 6316 to (33.46, -55.07, -116.37) mm, rotated rx 81.04 ry 30.21 rz 20.91 deg; joints [-6.114, -16.455, 80.193, 101.261, 107.446, 52.297, -153.967]
  MoveL 6317 to (35.18, -55.96, -117.93) mm, rotated rx 81.04 ry 30.21 rz 20.91 deg; joints [-6.187, -16.405, 80.05, 101.226, 107.459, 52.4, -153.967]
  MoveL 6318 to (32.86, -56.42, -118.06) mm, rotated rx 81.04 ry 30.21 rz 20.91 deg; joints [-6.113, -16.349, 79.934, 101.309, 107.415, 52.454, -153.967]
  MoveL 6319 to (30.67, -56.83, -118.17) mm, rotated rx 81.04 ry 30.21 rz 20.91 deg; joints [-6.042, -16.296, 79.826, 101.387, 107.373, 52.503, -153.967]
  MoveL 6320 to (28.55, -57.25, -118.33) mm, rotated rx 81.04 ry 30.21 rz 20.91 deg; joints [-5.974, -16.241, 79.716, 101.463, 107.333, 52.555, -153.967]
  MoveL 6321 to (26.46, -57.66, -118.44) mm, rotated rx 81.04 ry 30.21 rz 20.91 deg; joints [-5.907, -16.19, 79.612, 101.537, 107.293, 52.603, -153.967]
  MoveL 6322 to (24.36, -58.06, -118.55) mm, rotated rx 81.04 ry 30.21 rz 20.91 deg; joints [-5.84, -16.139, 79.507, 101.611, 107.253, 52.651, -153.967]
  MoveL 6323 to (22.26, -58.47, -118.77) mm, rotated rx 81.04 ry 30.21 rz 20.91 deg; joints [-5.774, -16.08, 79.39, 101.686, 107.212, 52.704, -153.967]
  MoveL 6324 to (20.16, -58.87, -118.99) mm, rotated rx 81.04 ry 30.21 rz 20.91 deg; joints [-5.709, -16.021, 79.273, 101.761, 107.171, 52.758, -153.967]
  MoveL 6325 to (18.07, -59.26, -119.11) mm, rotated rx 81.04 ry 30.21 rz 20.91 deg; joints [-5.642, -15.968, 79.167, 101.835, 107.131, 52.806, -153.967]
  MoveL 6326 to (15.97, -59.65, -119.11) mm, rotated rx 81.04 ry 30.21 rz 20.91 deg; joints [-5.573, -15.923, 79.073, 101.908, 107.091, 52.85, -153.967]
  MoveL 6327 to (13.87, -60.04, -119.22) mm, rotated rx 81.04 ry 30.21 rz 20.91 deg; joints [-5.506, -15.871, 78.967, 101.982, 107.05, 52.898, -153.967]
  MoveL 6328 to (11.74, -60.43, -119.42) mm, rotated rx 81.04 ry 30.21 rz 20.91 deg; joints [-5.44, -15.811, 78.849, 102.057, 107.008, 52.951, -153.967]
  MoveL 6329 to (9.76, -60.79, -119.6) mm, rotated rx 81.04 ry 30.21 rz 20.91 deg; joints [-5.378, -15.756, 78.741, 102.127, 106.97, 52.999, -153.967]
  MoveL 6330 to (7.93, -61.12, -119.82) mm, rotated rx 81.04 ry 30.21 rz 20.91 deg; joints [-5.321, -15.702, 78.635, 102.191, 106.934, 53.046, -153.967]
  MoveL 6331 to (6, -61.47, -119.91) mm, rotated rx 81.04 ry 30.21 rz 20.91 deg; joints [-5.26, -15.654, 78.537, 102.258, 106.896, 53.091, -153.967]
  MoveL 6332 to (3.94, -61.85, -119.92) mm, rotated rx 81.04 ry 30.21 rz 20.91 deg; joints [-5.193, -15.608, 78.441, 102.33, 106.856, 53.135, -153.967]
  MoveL 6333 to (1.27, -62.32, -120.02) mm, rotated rx 81.04 ry 30.21 rz 20.91 deg; joints [-5.108, -15.542, 78.309, 102.423, 106.803, 53.194, -153.967]
  MoveL 6334 to (-0.73, -62.66, -120.23) mm, rotated rx 81.04 ry 30.21 rz 20.91 deg; joints [-5.046, -15.483, 78.195, 102.493, 106.764, 53.244, -153.967]
  MoveL 6335 to (-2.91, -63.03, -120.43) mm, rotated rx 81.04 ry 30.21 rz 20.91 deg; joints [-4.978, -15.421, 78.075, 102.568, 106.721, 53.296, -153.967]
  MoveL 6336 to (-4.9, -63.35, -120.72) mm, rotated rx 81.04 ry 30.21 rz 20.91 deg; joints [-4.917, -15.357, 77.954, 102.637, 106.681, 53.348, -153.967]
  MoveL 6337 to (-6.86, -63.69, -120.85) mm, rotated rx 81.04 ry 30.21 rz 20.91 deg; joints [-4.856, -15.305, 77.849, 102.705, 106.642, 53.394, -153.967]
  MoveL 6338 to (-8.92, -64.06, -120.86) mm, rotated rx 81.04 ry 30.21 rz 20.91 deg; joints [-4.79, -15.257, 77.751, 102.776, 106.601, 53.439, -153.967]
  MoveL 6339 to (-10.67, -64.33, -121.09) mm, rotated rx 81.04 ry 30.21 rz 20.91 deg; joints [-4.737, -15.202, 77.647, 102.836, 106.566, 53.483, -153.967]
  Set speed (1000.0 mm/s)
  MoveL 6340 to (-32.01, -79.27, -121.09) mm, rotated rx 81.04 ry 30.21 rz 20.91 deg; joints [-4.054, -14.847, 76.056, 103.767, 105.968, 54.658, -153.967]
  Set speed (1000.0 mm/s)
  MoveL 6341 to (-35.76, -73.92, -132.28) mm, rotated rx 81.04 ry 30.21 rz 20.91 deg; joints [-4.07, -13.921, 74.974, 103.797, 105.938, 54.818, -153.967]
  Set speed (100.0 mm/s)
  MoveL 6342 to (-19.24, -62.35, -132.28) mm, rotated rx 81.04 ry 30.21 rz 20.91 deg; joints [-4.596, -14.204, 76.222, 103.08, 106.406, 53.902, -153.967]
  MoveL 6343 to (-17.11, -62.23, -132.28) mm, rotated rx 81.04 ry 30.21 rz 20.91 deg; joints [-4.663, -14.256, 76.311, 103.011, 106.446, 53.872, -153.967]
  MoveL 6344 to (-14.88, -62.13, -132.18) mm, rotated rx 81.04 ry 30.21 rz 20.91 deg; joints [-4.733, -14.318, 76.414, 102.94, 106.487, 53.838, -153.967]
  MoveL 6345 to (-12.53, -62.07, -131.89) mm, rotated rx 81.04 ry 30.21 rz 20.91 deg; joints [-4.805, -14.396, 76.54, 102.865, 106.53, 53.797, -153.967]
  MoveL 6346 to (-10.28, -62.01, -131.54) mm, rotated rx 81.04 ry 30.21 rz 20.91 deg; joints [-4.873, -14.475, 76.667, 102.793, 106.572, 53.755, -153.967]
  MoveL 6347 to (-8.22, -61.92, -131.35) mm, rotated rx 81.04 ry 30.21 rz 20.91 deg; joints [-4.937, -14.539, 76.771, 102.727, 106.61, 53.721, -153.967]
  MoveL 6348 to (-6.27, -61.83, -131.22) mm, rotated rx 81.04 ry 30.21 rz 20.91 deg; joints [-4.997, -14.595, 76.865, 102.664, 106.645, 53.689, -153.967]
  MoveL 6349 to (-4.22, -61.72, -131.17) mm, rotated rx 81.04 ry 30.21 rz 20.91 deg; joints [-5.062, -14.648, 76.954, 102.598, 106.683, 53.66, -153.967]
  MoveL 6350 to (-2.09, -61.61, -131.15) mm, rotated rx 81.04 ry 30.21 rz 20.91 deg; joints [-5.13, -14.701, 77.043, 102.529, 106.721, 53.63, -153.967]
  MoveL 6351 to (0.03, -61.5, -131.03) mm, rotated rx 81.04 ry 30.21 rz 20.91 deg; joints [-5.197, -14.76, 77.141, 102.461, 106.76, 53.597, -153.967]
  MoveL 6352 to (2.32, -61.38, -130.77) mm, rotated rx 81.04 ry 30.21 rz 20.91 deg; joints [-5.267, -14.832, 77.261, 102.386, 106.802, 53.556, -153.967]
  MoveL 6353 to (4.71, -61.25, -130.58) mm, rotated rx 81.04 ry 30.21 rz 20.91 deg; joints [-5.342, -14.902, 77.377, 102.309, 106.846, 53.517, -153.967]
  MoveL 6354 to (7.04, -61.11, -130.38) mm, rotated rx 81.04 ry 30.21 rz 20.91 deg; joints [-5.415, -14.971, 77.491, 102.233, 106.888, 53.477, -153.967]
  MoveL 6355 to (9.17, -60.99, -130.27) mm, rotated rx 81.04 ry 30.21 rz 20.91 deg; joints [-5.482, -15.029, 77.588, 102.164, 106.927, 53.444, -153.967]
  MoveL 6356 to (13.39, -60.74, -129.99) mm, rotated rx 81.04 ry 30.21 rz 20.91 deg; joints [-5.615, -15.147, 77.785, 102.026, 107.003, 53.377, -153.967]
  MoveL 6357 to (15.56, -60.61, -129.93) mm, rotated rx 81.04 ry 30.21 rz 20.91 deg; joints [-5.684, -15.202, 77.877, 101.956, 107.042, 53.346, -153.967]
  MoveL 6358 to (17.69, -60.46, -129.71) mm, rotated rx 81.04 ry 30.21 rz 20.91 deg; joints [-5.75, -15.266, 77.985, 101.886, 107.08, 53.308, -153.967]
  MoveL 6359 to (19.8, -60.32, -129.55) mm, rotated rx 81.04 ry 30.21 rz 20.91 deg; joints [-5.816, -15.326, 78.085, 101.817, 107.118, 53.273, -153.967]
  MoveL 6360 to (21.9, -60.17, -129.36) mm, rotated rx 81.04 ry 30.21 rz 20.91 deg; joints [-5.882, -15.387, 78.188, 101.747, 107.157, 53.237, -153.967]
  MoveL 6361 to (24.07, -60.03, -129.27) mm, rotated rx 81.04 ry 30.21 rz 20.91 deg; joints [-5.952, -15.443, 78.282, 101.676, 107.195, 53.205, -153.967]
  MoveL 6362 to (26.34, -59.87, -129.14) mm, rotated rx 81.04 ry 30.21 rz 20.91 deg; joints [-6.023, -15.504, 78.384, 101.602, 107.236, 53.169, -153.967]
  MoveL 6363 to (28.24, -59.77, -129.08) mm, rotated rx 81.04 ry 30.21 rz 20.91 deg; joints [-6.084, -15.552, 78.463, 101.54, 107.269, 53.144, -153.967]
  MoveL 6364 to (28.2, -59.11, -128.2) mm, rotated rx 81.04 ry 30.21 rz 20.91 deg; joints [-6.074, -15.601, 78.586, 101.526, 107.279, 53.066, -153.967]
  MoveL 6365 to (27.9, -58.91, -127.79) mm, rotated rx 81.04 ry 30.21 rz 20.91 deg; joints [-6.06, -15.619, 78.629, 101.531, 107.278, 53.039, -153.967]
  MoveL 6366 to (27.88, -58.84, -127.51) mm, rotated rx 81.04 ry 30.21 rz 20.91 deg; joints [-6.056, -15.636, 78.66, 101.53, 107.279, 53.024, -153.967]
  MoveL 6367 to (28.18, -58.97, -127.39) mm, rotated rx 81.04 ry 30.21 rz 20.91 deg; joints [-6.064, -15.653, 78.677, 101.523, 107.283, 53.025, -153.967]
  MoveL 6368 to (28.59, -59.16, -127.33) mm, rotated rx 81.04 ry 30.21 rz 20.91 deg; joints [-6.076, -15.669, 78.688, 101.514, 107.287, 53.032, -153.967]
  MoveL 6369 to (29.08, -59.43, -127.3) mm, rotated rx 81.04 ry 30.21 rz 20.91 deg; joints [-6.092, -15.687, 78.696, 101.503, 107.292, 53.043, -153.967]
  MoveL 6370 to (29.69, -59.76, -127.26) mm, rotated rx 81.04 ry 30.21 rz 20.91 deg; joints [-6.111, -15.708, 78.706, 101.491, 107.298, 53.057, -153.967]
  MoveL 6371 to (30.24, -60.07, -127.23) mm, rotated rx 81.04 ry 30.21 rz 20.91 deg; joints [-6.128, -15.727, 78.713, 101.479, 107.303, 53.071, -153.967]
  MoveL 6372 to (30.7, -60.34, -127.23) mm, rotated rx 81.04 ry 30.21 rz 20.91 deg; joints [-6.142, -15.742, 78.715, 101.471, 107.307, 53.085, -153.967]
  MoveL 6373 to (31.12, -60.58, -127.22) mm, rotated rx 81.04 ry 30.21 rz 20.91 deg; joints [-6.156, -15.756, 78.72, 101.462, 107.312, 53.096, -153.967]
  MoveL 6374 to (32.04, -61.06, -127.14) mm, rotated rx 81.04 ry 30.21 rz 20.91 deg; joints [-6.184, -15.79, 78.738, 101.442, 107.321, 53.115, -153.967]
  MoveL 6375 to (32.54, -61.32, -127.09) mm, rotated rx 81.04 ry 30.21 rz 20.91 deg; joints [-6.2, -15.808, 78.747, 101.432, 107.326, 53.126, -153.967]
  MoveL 6376 to (33, -61.54, -127.02) mm, rotated rx 81.04 ry 30.21 rz 20.91 deg; joints [-6.214, -15.827, 78.76, 101.422, 107.331, 53.133, -153.967]
  MoveL 6377 to (33.42, -61.73, -126.95) mm, rotated rx 81.04 ry 30.21 rz 20.91 deg; joints [-6.226, -15.845, 78.773, 101.412, 107.336, 53.139, -153.967]
  MoveL 6378 to (33.84, -61.93, -126.89) mm, rotated rx 81.04 ry 30.21 rz 20.91 deg; joints [-6.239, -15.861, 78.784, 101.403, 107.34, 53.146, -153.967]
  MoveL 6379 to (34.27, -62.16, -126.86) mm, rotated rx 81.04 ry 30.21 rz 20.91 deg; joints [-6.252, -15.877, 78.791, 101.394, 107.345, 53.156, -153.967]
  MoveL 6380 to (34.72, -62.42, -126.84) mm, rotated rx 81.04 ry 30.21 rz 20.91 deg; joints [-6.267, -15.892, 78.797, 101.385, 107.349, 53.167, -153.967]
  MoveL 6381 to (37.88, -64.29, -126.84) mm, rotated rx 81.04 ry 30.21 rz 20.91 deg; joints [-6.367, -15.992, 78.815, 101.323, 107.378, 53.261, -153.967]
  MoveL 6382 to (39.22, -65.21, -126.86) mm, rotated rx 81.04 ry 30.21 rz 20.91 deg; joints [-6.41, -16.035, 78.814, 101.3, 107.388, 53.31, -153.967]
  MoveL 6383 to (39.63, -65.61, -126.89) mm, rotated rx 81.04 ry 30.21 rz 20.91 deg; joints [-6.423, -16.048, 78.806, 101.295, 107.39, 53.333, -153.967]
  MoveL 6384 to (39.89, -65.96, -126.92) mm, rotated rx 81.04 ry 30.21 rz 20.91 deg; joints [-6.432, -16.057, 78.794, 101.294, 107.39, 53.355, -153.967]
  MoveL 6385 to (40.01, -66.28, -126.96) mm, rotated rx 81.04 ry 30.21 rz 20.91 deg; joints [-6.436, -16.061, 78.778, 101.297, 107.388, 53.376, -153.967]
  MoveL 6386 to (40.03, -66.43, -126.99) mm, rotated rx 81.04 ry 30.21 rz 20.91 deg; joints [-6.436, -16.061, 78.768, 101.299, 107.386, 53.386, -153.967]
  MoveL 6387 to (40.01, -66.57, -127.01) mm, rotated rx 81.04 ry 30.21 rz 20.91 deg; joints [-6.436, -16.061, 78.758, 101.303, 107.384, 53.396, -153.967]
  MoveL 6388 to (39.96, -66.7, -127.04) mm, rotated rx 81.04 ry 30.21 rz 20.91 deg; joints [-6.434, -16.06, 78.747, 101.307, 107.381, 53.406, -153.967]
  MoveL 6389 to (39.88, -66.82, -127.07) mm, rotated rx 81.04 ry 30.21 rz 20.91 deg; joints [-6.432, -16.058, 78.736, 101.312, 107.379, 53.416, -153.967]
  MoveL 6390 to (39.66, -67.04, -127.13) mm, rotated rx 81.04 ry 30.21 rz 20.91 deg; joints [-6.425, -16.052, 78.711, 101.323, 107.372, 53.434, -153.967]
  MoveL 6391 to (38.95, -67.39, -127.26) mm, rotated rx 81.04 ry 30.21 rz 20.91 deg; joints [-6.403, -16.031, 78.655, 101.353, 107.355, 53.468, -153.967]
  MoveL 6392 to (37.97, -67.66, -127.4) mm, rotated rx 81.04 ry 30.21 rz 20.91 deg; joints [-6.373, -16.002, 78.594, 101.389, 107.335, 53.498, -153.967]
  MoveL 6393 to (35.65, -67.96, -127.67) mm, rotated rx 81.04 ry 30.21 rz 20.91 deg; joints [-6.301, -15.933, 78.47, 101.468, 107.292, 53.548, -153.967]
  MoveL 6394 to (33.24, -68.12, -127.91) mm, rotated rx 81.04 ry 30.21 rz 20.91 deg; joints [-6.225, -15.862, 78.353, 101.546, 107.248, 53.588, -153.967]
  MoveL 6395 to (-20.65, -71.26, -132.99) mm, rotated rx 81.04 ry 30.21 rz 20.91 deg; joints [-4.557, -14.231, 75.643, 103.285, 106.25, 54.512, -153.967]
  MoveL 6396 to (-24.48, -71.48, -133.35) mm, rotated rx 81.04 ry 30.21 rz 20.91 deg; joints [-4.44, -14.111, 75.44, 103.408, 106.176, 54.583, -153.967]
  MoveL 6397 to (-28.22, -71.52, -133.77) mm, rotated rx 81.04 ry 30.21 rz 20.91 deg; joints [-4.326, -13.987, 75.242, 103.524, 106.106, 54.644, -153.967]
  MoveL 6398 to (-29.69, -71.26, -133.98) mm, rotated rx 81.04 ry 30.21 rz 20.91 deg; joints [-4.282, -13.931, 75.173, 103.565, 106.082, 54.652, -153.967]
  MoveL 6399 to (-30.18, -71.02, -134.07) mm, rotated rx 81.04 ry 30.21 rz 20.91 deg; joints [-4.268, -13.909, 75.155, 103.576, 106.077, 54.647, -153.967]
  MoveL 6400 to (-30.35, -70.87, -134.12) mm, rotated rx 81.04 ry 30.21 rz 20.91 deg; joints [-4.263, -13.9, 75.151, 103.579, 106.076, 54.641, -153.967]
  MoveL 6401 to (-30.46, -70.69, -134.16) mm, rotated rx 81.04 ry 30.21 rz 20.91 deg; joints [-4.26, -13.892, 75.151, 103.579, 106.076, 54.632, -153.967]
  MoveL 6402 to (-30.5, -70.49, -134.2) mm, rotated rx 81.04 ry 30.21 rz 20.91 deg; joints [-4.259, -13.886, 75.156, 103.577, 106.078, 54.621, -153.967]
  MoveL 6403 to (-30.48, -70.26, -134.23) mm, rotated rx 81.04 ry 30.21 rz 20.91 deg; joints [-4.26, -13.881, 75.165, 103.572, 106.082, 54.608, -153.967]
  MoveL 6404 to (-30.38, -70, -134.26) mm, rotated rx 81.04 ry 30.21 rz 20.91 deg; joints [-4.264, -13.879, 75.179, 103.564, 106.088, 54.591, -153.967]
  MoveL 6405 to (-30.2, -69.7, -134.29) mm, rotated rx 81.04 ry 30.21 rz 20.91 deg; joints [-4.27, -13.878, 75.198, 103.554, 106.095, 54.572, -153.967]
  MoveL 6406 to (-28.61, -68.2, -134.33) mm, rotated rx 81.04 ry 30.21 rz 20.91 deg; joints [-4.321, -13.898, 75.333, 103.478, 106.146, 54.461, -153.967]
  MoveL 6407 to (-26.93, -66.94, -134.33) mm, rotated rx 81.04 ry 30.21 rz 20.91 deg; joints [-4.374, -13.925, 75.465, 103.404, 106.195, 54.362, -153.967]
  MoveL 6408 to (-23.64, -65.04, -134.38) mm, rotated rx 81.04 ry 30.21 rz 20.91 deg; joints [-4.48, -13.983, 75.687, 103.268, 106.282, 54.207, -153.967]
  MoveL 6409 to (-20.26, -63.98, -134.49) mm, rotated rx 81.04 ry 30.21 rz 20.91 deg; joints [-4.589, -14.048, 75.863, 103.144, 106.357, 54.108, -153.967]
  MoveL 6410 to (-14.22, -63.62, -134.79) mm, rotated rx 81.04 ry 30.21 rz 20.91 deg; joints [-4.785, -14.177, 76.086, 102.95, 106.468, 54.033, -153.967]
  MoveL 6411 to (-11.88, -63.98, -134.92) mm, rotated rx 81.04 ry 30.21 rz 20.91 deg; joints [-4.86, -14.231, 76.146, 102.884, 106.504, 54.036, -153.967]
  MoveL 6412 to (22.24, -70.68, -136.78) mm, rotated rx 81.04 ry 30.21 rz 20.91 deg; joints [-5.969, -15.031, 76.892, 101.956, 107.003, 54.208, -153.967]
  MoveL 6413 to (25.16, -71.24, -136.94) mm, rotated rx 81.04 ry 30.21 rz 20.91 deg; joints [-6.063, -15.097, 76.952, 101.877, 107.045, 54.224, -153.967]
  MoveL 6414 to (28.88, -71.49, -137.19) mm, rotated rx 81.04 ry 30.21 rz 20.91 deg; joints [-6.186, -15.174, 77.047, 101.767, 107.105, 54.217, -153.967]
  MoveL 6415 to (30.35, -71.26, -137.33) mm, rotated rx 81.04 ry 30.21 rz 20.91 deg; joints [-6.234, -15.196, 77.096, 101.718, 107.133, 54.195, -153.967]
  MoveL 6416 to (30.84, -71.02, -137.4) mm, rotated rx 81.04 ry 30.21 rz 20.91 deg; joints [-6.251, -15.2, 77.118, 101.698, 107.145, 54.178, -153.967]
  MoveL 6417 to (31, -70.86, -137.43) mm, rotated rx 81.04 ry 30.21 rz 20.91 deg; joints [-6.257, -15.2, 77.128, 101.69, 107.149, 54.168, -153.967]
  MoveL 6418 to (31.11, -70.68, -137.47) mm, rotated rx 81.04 ry 30.21 rz 20.91 deg; joints [-6.261, -15.198, 77.137, 101.683, 107.154, 54.157, -153.967]
  MoveL 6419 to (31.15, -70.48, -137.5) mm, rotated rx 81.04 ry 30.21 rz 20.91 deg; joints [-6.263, -15.194, 77.145, 101.678, 107.157, 54.145, -153.967]
  MoveL 6420 to (31.13, -70.24, -137.54) mm, rotated rx 81.04 ry 30.21 rz 20.91 deg; joints [-6.263, -15.188, 77.152, 101.674, 107.159, 54.132, -153.967]
  MoveL 6421 to (31.03, -69.98, -137.57) mm, rotated rx 81.04 ry 30.21 rz 20.91 deg; joints [-6.26, -15.18, 77.158, 101.672, 107.161, 54.117, -153.967]
  MoveL 6422 to (30.85, -69.69, -137.61) mm, rotated rx 81.04 ry 30.21 rz 20.91 deg; joints [-6.255, -15.17, 77.163, 101.672, 107.162, 54.101, -153.967]
  MoveL 6423 to (29.23, -68.21, -137.73) mm, rotated rx 81.04 ry 30.21 rz 20.91 deg; joints [-6.206, -15.104, 77.166, 101.693, 107.153, 54.025, -153.967]
  MoveL 6424 to (28.82, -67.9, -137.75) mm, rotated rx 81.04 ry 30.21 rz 20.91 deg; joints [-6.193, -15.088, 77.164, 101.7, 107.15, 54.01, -153.967]
  MoveL 6425 to (28.43, -67.65, -137.8) mm, rotated rx 81.04 ry 30.21 rz 20.91 deg; joints [-6.181, -15.073, 77.158, 101.707, 107.147, 53.999, -153.967]
  MoveL 6426 to (28.05, -67.42, -137.87) mm, rotated rx 81.04 ry 30.21 rz 20.91 deg; joints [-6.17, -15.056, 77.148, 101.714, 107.143, 53.991, -153.967]
  MoveL 6427 to (27.68, -67.19, -137.93) mm, rotated rx 81.04 ry 30.21 rz 20.91 deg; joints [-6.159, -15.04, 77.14, 101.721, 107.139, 53.982, -153.967]
  MoveL 6428 to (27.3, -66.92, -137.96) mm, rotated rx 81.04 ry 30.21 rz 20.91 deg; joints [-6.147, -15.025, 77.136, 101.728, 107.136, 53.97, -153.967]
  MoveL 6429 to (23.6, -64.05, -137.97) mm, rotated rx 81.04 ry 30.21 rz 20.91 deg; joints [-6.031, -14.898, 77.145, 101.787, 107.111, 53.819, -153.967]
  MoveL 6430 to (23.24, -63.79, -137.99) mm, rotated rx 81.04 ry 30.21 rz 20.91 deg; joints [-6.02, -14.885, 77.142, 101.793, 107.108, 53.807, -153.967]
  MoveL 6431 to (22.86, -63.5, -138) mm, rotated rx 81.04 ry 30.21 rz 20.91 deg; joints [-6.008, -14.871, 77.142, 101.799, 107.105, 53.792, -153.967]
  MoveL 6432 to (22.04, -62.86, -138) mm, rotated rx 81.04 ry 30.21 rz 20.91 deg; joints [-5.982, -14.843, 77.143, 101.812, 107.1, 53.759, -153.967]
  MoveL 6433 to (21.58, -62.52, -138.01) mm, rotated rx 81.04 ry 30.21 rz 20.91 deg; joints [-5.968, -14.827, 77.143, 101.82, 107.096, 53.742, -153.967]
  MoveL 6434 to (21.09, -62.18, -138.03) mm, rotated rx 81.04 ry 30.21 rz 20.91 deg; joints [-5.953, -14.809, 77.14, 101.828, 107.092, 53.725, -153.967]
  MoveL 6435 to (20.53, -61.83, -138.06) mm, rotated rx 81.04 ry 30.21 rz 20.91 deg; joints [-5.935, -14.789, 77.134, 101.839, 107.087, 53.71, -153.967]
  MoveL 6436 to (19.93, -61.55, -138.08) mm, rotated rx 81.04 ry 30.21 rz 20.91 deg; joints [-5.916, -14.769, 77.123, 101.853, 107.08, 53.698, -153.967]
  MoveL 6437 to (19.31, -61.32, -138.1) mm, rotated rx 81.04 ry 30.21 rz 20.91 deg; joints [-5.897, -14.75, 77.11, 101.867, 107.073, 53.69, -153.967]
  MoveL 6438 to (20.41, -62.04, -139.08) mm, rotated rx 81.04 ry 30.21 rz 20.91 deg; joints [-5.943, -14.72, 77.01, 101.849, 107.079, 53.766, -153.967]
  MoveL 6439 to (19.09, -62.27, -139.5) mm, rotated rx 81.04 ry 30.21 rz 20.91 deg; joints [-5.905, -14.662, 76.905, 101.896, 107.053, 53.81, -153.967]
  MoveL 6440 to (17.6, -62.38, -139.82) mm, rotated rx 81.04 ry 30.21 rz 20.91 deg; joints [-5.861, -14.606, 76.811, 101.945, 107.025, 53.845, -153.967]
  MoveL 6441 to (15.91, -62.4, -140.06) mm, rotated rx 81.04 ry 30.21 rz 20.91 deg; joints [-5.809, -14.549, 76.723, 101.999, 106.994, 53.872, -153.967]
  MoveL 6442 to (13.78, -62.3, -140.28) mm, rotated rx 81.04 ry 30.21 rz 20.91 deg; joints [-5.743, -14.481, 76.626, 102.063, 106.958, 53.894, -153.967]
  MoveL 6443 to (11.65, -62.17, -140.39) mm, rotated rx 81.04 ry 30.21 rz 20.91 deg; joints [-5.676, -14.419, 76.541, 102.127, 106.923, 53.911, -153.967]
  MoveL 6444 to (9.52, -62.03, -140.5) mm, rotated rx 81.04 ry 30.21 rz 20.91 deg; joints [-5.609, -14.358, 76.456, 102.191, 106.887, 53.928, -153.967]
  MoveL 6445 to (7.38, -61.92, -140.73) mm, rotated rx 81.04 ry 30.21 rz 20.91 deg; joints [-5.544, -14.288, 76.358, 102.256, 106.851, 53.951, -153.967]
  MoveL 6446 to (5.26, -61.78, -140.85) mm, rotated rx 81.04 ry 30.21 rz 20.91 deg; joints [-5.477, -14.226, 76.272, 102.32, 106.816, 53.968, -153.967]
  MoveL 6447 to (3.13, -61.65, -141.08) mm, rotated rx 81.04 ry 30.21 rz 20.91 deg; joints [-5.412, -14.156, 76.173, 102.384, 106.78, 53.991, -153.967]
  MoveL 6448 to (1, -61.5, -141.2) mm, rotated rx 81.04 ry 30.21 rz 20.91 deg; joints [-5.345, -14.093, 76.087, 102.448, 106.744, 54.008, -153.967]
  MoveL 6449 to (-1.13, -61.36, -141.31) mm, rotated rx 81.04 ry 30.21 rz 20.91 deg; joints [-5.279, -14.031, 76, 102.511, 106.708, 54.025, -153.967]
  MoveL 6450 to (-3.26, -61.21, -141.55) mm, rotated rx 81.04 ry 30.21 rz 20.91 deg; joints [-5.214, -13.96, 75.9, 102.575, 106.672, 54.047, -153.967]
  MoveL 6451 to (-5.3, -61.05, -141.65) mm, rotated rx 81.04 ry 30.21 rz 20.91 deg; joints [-5.15, -13.9, 75.818, 102.636, 106.638, 54.063, -153.967]
  MoveL 6452 to (-7.28, -60.9, -141.86) mm, rotated rx 81.04 ry 30.21 rz 20.91 deg; joints [-5.089, -13.834, 75.727, 102.695, 106.605, 54.082, -153.967]
  MoveL 6453 to (-9.64, -60.73, -142.02) mm, rotated rx 81.04 ry 30.21 rz 20.91 deg; joints [-5.016, -13.761, 75.626, 102.766, 106.565, 54.104, -153.967]
  MoveL 6454 to (-12.36, -60.51, -142.11) mm, rotated rx 81.04 ry 30.21 rz 20.91 deg; joints [-4.931, -13.684, 75.522, 102.846, 106.519, 54.122, -153.967]
  MoveL 6455 to (-14.43, -60.36, -142.17) mm, rotated rx 81.04 ry 30.21 rz 20.91 deg; joints [-4.866, -13.626, 75.441, 102.908, 106.484, 54.138, -153.967]
  MoveL 6456 to (-16.35, -60.22, -142.3) mm, rotated rx 81.04 ry 30.21 rz 20.91 deg; joints [-4.806, -13.566, 75.358, 102.965, 106.452, 54.155, -153.967]
  MoveL 6457 to (-18.32, -60.07, -142.41) mm, rotated rx 81.04 ry 30.21 rz 20.91 deg; joints [-4.745, -13.507, 75.276, 103.024, 106.418, 54.171, -153.967]
  MoveL 6458 to (-20.27, -59.91, -142.52) mm, rotated rx 81.04 ry 30.21 rz 20.91 deg; joints [-4.684, -13.448, 75.194, 103.082, 106.385, 54.188, -153.967]
  MoveL 6459 to (-22.32, -59.76, -142.59) mm, rotated rx 81.04 ry 30.21 rz 20.91 deg; joints [-4.62, -13.389, 75.112, 103.143, 106.351, 54.204, -153.967]
  MoveL 6460 to (-24.54, -59.58, -142.69) mm, rotated rx 81.04 ry 30.21 rz 20.91 deg; joints [-4.551, -13.323, 75.021, 103.209, 106.313, 54.221, -153.967]
  MoveL 6461 to (-26.94, -59.35, -142.95) mm, rotated rx 81.04 ry 30.21 rz 20.91 deg; joints [-4.478, -13.241, 74.907, 103.28, 106.272, 54.245, -153.967]
  MoveL 6462 to (-29.15, -59.68, -143.93) mm, rotated rx 81.04 ry 30.21 rz 20.91 deg; joints [-4.419, -13.12, 74.693, 103.356, 106.223, 54.333, -153.967]
  MoveL 6463 to (-28.15, -59.12, -144.42) mm, rotated rx 81.04 ry 30.21 rz 20.91 deg; joints [-4.457, -13.105, 74.708, 103.316, 106.248, 54.307, -153.967]
  MoveL 6464 to (-27.63, -58.83, -144.73) mm, rotated rx 81.04 ry 30.21 rz 20.91 deg; joints [-4.477, -13.094, 74.71, 103.295, 106.26, 54.296, -153.967]
  MoveL 6465 to (-27.55, -58.77, -144.88) mm, rotated rx 81.04 ry 30.21 rz 20.91 deg; joints [-4.481, -13.085, 74.699, 103.292, 106.262, 54.298, -153.967]
  MoveL 6466 to (-27.86, -58.94, -144.92) mm, rotated rx 81.04 ry 30.21 rz 20.91 deg; joints [-4.472, -13.076, 74.675, 103.304, 106.254, 54.314, -153.967]
  MoveL 6467 to (-28.26, -59.16, -144.93) mm, rotated rx 81.04 ry 30.21 rz 20.91 deg; joints [-4.459, -13.068, 74.645, 103.321, 106.243, 54.333, -153.967]
  MoveL 6468 to (-28.69, -59.38, -144.97) mm, rotated rx 81.04 ry 30.21 rz 20.91 deg; joints [-4.446, -13.057, 74.613, 103.338, 106.232, 54.353, -153.967]
  MoveL 6469 to (-29.1, -59.58, -145.03) mm, rotated rx 81.04 ry 30.21 rz 20.91 deg; joints [-4.434, -13.045, 74.58, 103.354, 106.222, 54.373, -153.967]
  MoveL 6470 to (-29.51, -59.78, -145.07) mm, rotated rx 81.04 ry 30.21 rz 20.91 deg; joints [-4.421, -13.034, 74.548, 103.371, 106.211, 54.392, -153.967]
  MoveL 6471 to (-29.94, -60.02, -145.09) mm, rotated rx 81.04 ry 30.21 rz 20.91 deg; joints [-4.408, -13.024, 74.517, 103.388, 106.2, 54.413, -153.967]
  MoveL 6472 to (-32.22, -61.32, -145.09) mm, rotated rx 81.04 ry 30.21 rz 20.91 deg; joints [-4.336, -12.981, 74.359, 103.482, 106.139, 54.521, -153.967]
  MoveL 6473 to (-32.62, -61.53, -145.11) mm, rotated rx 81.04 ry 30.21 rz 20.91 deg; joints [-4.323, -12.972, 74.329, 103.498, 106.129, 54.541, -153.967]
  MoveL 6474 to (-32.97, -61.7, -145.14) mm, rotated rx 81.04 ry 30.21 rz 20.91 deg; joints [-4.313, -12.962, 74.302, 103.512, 106.12, 54.557, -153.967]
  MoveL 6475 to (-33.38, -61.92, -145.16) mm, rotated rx 81.04 ry 30.21 rz 20.91 deg; joints [-4.3, -12.953, 74.272, 103.529, 106.109, 54.576, -153.967]
  MoveL 6476 to (-33.9, -62.2, -145.18) mm, rotated rx 81.04 ry 30.21 rz 20.91 deg; joints [-4.284, -12.941, 74.234, 103.55, 106.095, 54.601, -153.967]
  MoveL 6477 to (-34.55, -62.52, -145.24) mm, rotated rx 81.04 ry 30.21 rz 20.91 deg; joints [-4.264, -12.925, 74.185, 103.576, 106.078, 54.631, -153.967]
  MoveL 6478 to (-35.09, -62.81, -145.27) mm, rotated rx 81.04 ry 30.21 rz 20.91 deg; joints [-4.247, -12.912, 74.145, 103.598, 106.064, 54.657, -153.967]
  MoveL 6479 to (-35.56, -63.08, -145.27) mm, rotated rx 81.04 ry 30.21 rz 20.91 deg; joints [-4.232, -12.903, 74.112, 103.617, 106.051, 54.679, -153.967]
  MoveL 6480 to (-36.92, -63.86, -145.27) mm, rotated rx 81.04 ry 30.21 rz 20.91 deg; joints [-4.189, -12.876, 74.016, 103.672, 106.015, 54.745, -153.967]
  MoveL 6481 to (-39.58, -65.04, -145.61) mm, rotated rx 81.04 ry 30.21 rz 20.91 deg; joints [-4.109, -12.797, 73.807, 103.776, 105.947, 54.866, -153.967]
  MoveL 6482 to (-40.85, -65.33, -146.04) mm, rotated rx 81.04 ry 30.21 rz 20.91 deg; joints [-4.075, -12.737, 73.692, 103.82, 105.917, 54.918, -153.967]
  MoveL 6483 to (-42.06, -65.44, -146.64) mm, rotated rx 81.04 ry 30.21 rz 20.91 deg; joints [-4.043, -12.665, 73.569, 103.86, 105.89, 54.965, -153.967]
  MoveL 6484 to (-44.35, -65.05, -148.35) mm, rotated rx 81.04 ry 30.21 rz 20.91 deg; joints [-3.992, -12.481, 73.302, 103.927, 105.846, 55.043, -153.967]
  MoveL 6485 to (-46.45, -63.88, -150.75) mm, rotated rx 81.04 ry 30.21 rz 20.91 deg; joints [-3.955, -12.244, 73.005, 103.975, 105.814, 55.099, -153.967]
  MoveL 6486 to (-47.84, -62.36, -153.14) mm, rotated rx 81.04 ry 30.21 rz 20.91 deg; joints [-3.94, -12.022, 72.754, 103.995, 105.8, 55.126, -153.967]
  MoveL 6487 to (-48.07, -61.63, -154.08) mm, rotated rx 81.04 ry 30.21 rz 20.91 deg; joints [-3.944, -11.942, 72.675, 103.991, 105.802, 55.125, -153.967]
  MoveL 6488 to (-47.99, -60.92, -154.85) mm, rotated rx 81.04 ry 30.21 rz 20.91 deg; joints [-3.955, -11.881, 72.628, 103.978, 105.811, 55.114, -153.967]
  MoveL 6489 to (-47.84, -60.58, -155.17) mm, rotated rx 81.04 ry 30.21 rz 20.91 deg; joints [-3.964, -11.859, 72.616, 103.968, 105.817, 55.105, -153.967]
  MoveL 6490 to (-47.61, -60.24, -155.45) mm, rotated rx 81.04 ry 30.21 rz 20.91 deg; joints [-3.975, -11.842, 72.611, 103.955, 105.825, 55.093, -153.967]
  MoveL 6491 to (-46.91, -59.58, -155.88) mm, rotated rx 81.04 ry 30.21 rz 20.91 deg; joints [-4.002, -11.823, 72.627, 103.923, 105.846, 55.062, -153.967]
  MoveL 6492 to (-45.91, -58.94, -156.14) mm, rotated rx 81.04 ry 30.21 rz 20.91 deg; joints [-4.036, -11.824, 72.673, 103.882, 105.874, 55.02, -153.967]
  MoveL 6493 to (-44.6, -58.33, -156.22) mm, rotated rx 81.04 ry 30.21 rz 20.91 deg; joints [-4.078, -11.846, 72.751, 103.831, 105.907, 54.969, -153.967]
  MoveL 6494 to (-44.11, -58.13, -156.22) mm, rotated rx 81.04 ry 30.21 rz 20.91 deg; joints [-4.094, -11.856, 72.782, 103.812, 105.919, 54.95, -153.967]
  MoveL 6495 to (-43.69, -57.99, -156.17) mm, rotated rx 81.04 ry 30.21 rz 20.91 deg; joints [-4.106, -11.87, 72.812, 103.797, 105.929, 54.934, -153.967]
  MoveL 6496 to (-43.28, -57.87, -156.11) mm, rotated rx 81.04 ry 30.21 rz 20.91 deg; joints [-4.118, -11.883, 72.843, 103.782, 105.939, 54.919, -153.967]
  MoveL 6497 to (-42.83, -57.71, -156.07) mm, rotated rx 81.04 ry 30.21 rz 20.91 deg; joints [-4.132, -11.896, 72.874, 103.765, 105.95, 54.901, -153.967]
  MoveL 6498 to (-42.36, -57.53, -156.05) mm, rotated rx 81.04 ry 30.21 rz 20.91 deg; joints [-4.147, -11.908, 72.905, 103.748, 105.961, 54.884, -153.967]
  MoveL 6499 to (-41.87, -57.33, -156.05) mm, rotated rx 81.04 ry 30.21 rz 20.91 deg; joints [-4.162, -11.919, 72.937, 103.729, 105.973, 54.865, -153.967]
  MoveL 6500 to (-41.39, -57.13, -156.05) mm, rotated rx 81.04 ry 30.21 rz 20.91 deg; joints [-4.177, -11.929, 72.967, 103.711, 105.985, 54.846, -153.967]
  MoveL 6501 to (-40.92, -56.93, -156.06) mm, rotated rx 81.04 ry 30.21 rz 20.91 deg; joints [-4.192, -11.938, 72.995, 103.693, 105.997, 54.828, -153.967]
  MoveL 6502 to (-40.47, -56.73, -156.07) mm, rotated rx 81.04 ry 30.21 rz 20.91 deg; joints [-4.207, -11.947, 73.023, 103.675, 106.008, 54.811, -153.967]
  MoveL 6503 to (-40.04, -56.57, -156.05) mm, rotated rx 81.04 ry 30.21 rz 20.91 deg; joints [-4.22, -11.957, 73.052, 103.659, 106.019, 54.794, -153.967]
  MoveL 6504 to (-39.6, -56.41, -156.01) mm, rotated rx 81.04 ry 30.21 rz 20.91 deg; joints [-4.233, -11.97, 73.083, 103.643, 106.029, 54.777, -153.967]
  MoveL 6505 to (-39.08, -56.23, -155.96) mm, rotated rx 81.04 ry 30.21 rz 20.91 deg; joints [-4.249, -11.985, 73.119, 103.624, 106.042, 54.758, -153.967]
  MoveL 6506 to (-38.42, -56.01, -155.91) mm, rotated rx 81.04 ry 30.21 rz 20.91 deg; joints [-4.269, -12.003, 73.164, 103.599, 106.057, 54.733, -153.967]
  MoveL 6507 to (-37.81, -55.78, -155.89) mm, rotated rx 81.04 ry 30.21 rz 20.91 deg; joints [-4.288, -12.018, 73.204, 103.576, 106.072, 54.71, -153.967]
  MoveL 6508 to (-35.39, -54.78, -155.89) mm, rotated rx 81.04 ry 30.21 rz 20.91 deg; joints [-4.364, -12.07, 73.355, 103.484, 106.131, 54.618, -153.967]
  MoveL 6509 to (-34.81, -54.56, -155.85) mm, rotated rx 81.04 ry 30.21 rz 20.91 deg; joints [-4.382, -12.085, 73.395, 103.462, 106.145, 54.595, -153.967]
  MoveL 6510 to (-34.28, -54.37, -155.79) mm, rotated rx 81.04 ry 30.21 rz 20.91 deg; joints [-4.398, -12.1, 73.433, 103.442, 106.158, 54.574, -153.967]
  MoveL 6511 to (-34.08, -54.31, -155.64) mm, rotated rx 81.04 ry 30.21 rz 20.91 deg; joints [-4.403, -12.115, 73.461, 103.434, 106.163, 54.561, -153.967]
  MoveL 6512 to (-34.2, -54.35, -155.38) mm, rotated rx 81.04 ry 30.21 rz 20.91 deg; joints [-4.396, -12.131, 73.484, 103.438, 106.162, 54.554, -153.967]
  MoveL 6513 to (-34.63, -54.49, -154.97) mm, rotated rx 81.04 ry 30.21 rz 20.91 deg; joints [-4.378, -12.15, 73.504, 103.453, 106.153, 54.55, -153.967]
  MoveL 6514 to (-33.96, -55.27, -154.17) mm, rotated rx 81.04 ry 30.21 rz 20.91 deg; joints [-4.389, -12.232, 73.582, 103.445, 106.158, 54.556, -153.967]
  MoveL 6515 to (-32.03, -55.72, -153.95) mm, rotated rx 81.04 ry 30.21 rz 20.91 deg; joints [-4.447, -12.303, 73.664, 103.392, 106.187, 54.551, -153.967]
  MoveL 6516 to (-30.07, -56.15, -153.79) mm, rotated rx 81.04 ry 30.21 rz 20.91 deg; joints [-4.507, -12.371, 73.741, 103.339, 106.217, 54.549, -153.967]
  MoveL 6517 to (-28.06, -56.58, -153.64) mm, rotated rx 81.04 ry 30.21 rz 20.91 deg; joints [-4.569, -12.439, 73.819, 103.284, 106.248, 54.546, -153.967]
  MoveL 6518 to (-26.23, -56.99, -153.35) mm, rotated rx 81.04 ry 30.21 rz 20.91 deg; joints [-4.623, -12.511, 73.906, 103.234, 106.277, 54.537, -153.967]
  MoveL 6519 to (-24.17, -57.43, -153.16) mm, rotated rx 81.04 ry 30.21 rz 20.91 deg; joints [-4.686, -12.583, 73.989, 103.178, 106.309, 54.533, -153.967]
  MoveL 6520 to (-22, -57.9, -152.98) mm, rotated rx 81.04 ry 30.21 rz 20.91 deg; joints [-4.752, -12.657, 74.073, 103.119, 106.342, 54.53, -153.967]
  MoveL 6521 to (-19.81, -58.36, -152.89) mm, rotated rx 81.04 ry 30.21 rz 20.91 deg; joints [-4.821, -12.725, 74.149, 103.059, 106.376, 54.53, -153.967]
  MoveL 6522 to (-17.13, -58.91, -152.8) mm, rotated rx 81.04 ry 30.21 rz 20.91 deg; joints [-4.904, -12.807, 74.238, 102.986, 106.416, 54.532, -153.967]
  MoveL 6523 to (-15.21, -59.3, -152.69) mm, rotated rx 81.04 ry 30.21 rz 20.91 deg; joints [-4.963, -12.868, 74.307, 102.933, 106.446, 54.53, -153.967]
  MoveL 6524 to (-13.42, -59.66, -152.48) mm, rotated rx 81.04 ry 30.21 rz 20.91 deg; joints [-5.017, -12.933, 74.384, 102.884, 106.474, 54.524, -153.967]
  MoveL 6525 to (-11.45, -60.06, -152.29) mm, rotated rx 81.04 ry 30.21 rz 20.91 deg; joints [-5.078, -13.001, 74.463, 102.83, 106.504, 54.52, -153.967]
  MoveL 6526 to (-9.35, -60.48, -152.17) mm, rotated rx 81.04 ry 30.21 rz 20.91 deg; joints [-5.143, -13.067, 74.538, 102.773, 106.536, 54.519, -153.967]
  MoveL 6527 to (-7.28, -60.89, -151.99) mm, rotated rx 81.04 ry 30.21 rz 20.91 deg; joints [-5.206, -13.137, 74.618, 102.716, 106.568, 54.515, -153.967]
  MoveL 6528 to (-5.21, -61.3, -151.87) mm, rotated rx 81.04 ry 30.21 rz 20.91 deg; joints [-5.27, -13.203, 74.692, 102.659, 106.6, 54.513, -153.967]
  MoveL 6529 to (-3.07, -61.71, -151.69) mm, rotated rx 81.04 ry 30.21 rz 20.91 deg; joints [-5.336, -13.274, 74.774, 102.6, 106.633, 54.509, -153.967]
  MoveL 6530 to (-0.97, -62.12, -151.57) mm, rotated rx 81.04 ry 30.21 rz 20.91 deg; joints [-5.401, -13.34, 74.848, 102.543, 106.665, 54.508, -153.967]
  MoveL 6531 to (1.13, -62.51, -151.34) mm, rotated rx 81.04 ry 30.21 rz 20.91 deg; joints [-5.465, -13.413, 74.935, 102.484, 106.697, 54.501, -153.967]
  MoveL 6532 to (3.23, -62.91, -151.23) mm, rotated rx 81.04 ry 30.21 rz 20.91 deg; joints [-5.53, -13.478, 75.007, 102.427, 106.729, 54.501, -153.967]
  MoveL 6533 to (5.32, -63.31, -151.11) mm, rotated rx 81.04 ry 30.21 rz 20.91 deg; joints [-5.595, -13.543, 75.08, 102.369, 106.761, 54.5, -153.967]
  MoveL 6534 to (7.43, -63.69, -150.89) mm, rotated rx 81.04 ry 30.21 rz 20.91 deg; joints [-5.66, -13.615, 75.166, 102.311, 106.794, 54.493, -153.967]
  MoveL 6535 to (9.34, -63.98, -150.68) mm, rotated rx 81.04 ry 30.21 rz 20.91 deg; joints [-5.718, -13.68, 75.246, 102.257, 106.825, 54.484, -153.967]
  MoveL 6536 to (11.09, -64.18, -150.39) mm, rotated rx 81.04 ry 30.21 rz 20.91 deg; joints [-5.77, -13.746, 75.333, 102.206, 106.854, 54.467, -153.967]
  MoveL 6537 to (12.72, -64.29, -149.99) mm, rotated rx 81.04 ry 30.21 rz 20.91 deg; joints [-5.818, -13.815, 75.433, 102.157, 106.882, 54.441, -153.967]
  MoveL 6538 to (11.45, -63.5, -149.06) mm, rotated rx 81.04 ry 30.21 rz 20.91 deg; joints [-5.768, -13.838, 75.527, 102.178, 106.874, 54.363, -153.967]
  MoveL 6539 to (11.99, -63.73, -149.05) mm, rotated rx 81.04 ry 30.21 rz 20.91 deg; joints [-5.784, -13.855, 75.536, 102.166, 106.88, 54.372, -153.967]
  MoveL 6540 to (12.46, -63.97, -149.03) mm, rotated rx 81.04 ry 30.21 rz 20.91 deg; joints [-5.799, -13.871, 75.545, 102.156, 106.885, 54.382, -153.967]
